LIN {X 0,Y 248.183,Z 542.153,A -85,B 0,C 180,E1 -18821.434,E2 -18821.434} C_VEL
LIN {X 0,Y 249.329,Z 538.255,A -85,B 0,C 180,E1 -18823.863,E2 -18823.863} C_VEL
LIN {X 0,Y 251.024,Z 533.251,A -85,B 0,C 180,E1 -18826.259,E2 -18826.259} C_VEL
LIN {X 0,Y 253.003,Z 526.994,A -85,B 0,C 180,E1 -18828.63,E2 -18828.63} C_VEL
LIN {X 0,Y 255.334,Z 519.2,A -85,B 0,C 180,E1 -18830.967,E2 -18830.967} C_VEL
LIN {X 0,Y 258.267,Z 509.494,A -85,B 0,C 180,E1 -18833.24,E2 -18833.24} C_VEL
LIN {X 0,Y 261.068,Z 499.47,A -85,B 0,C 180,E1 -18835.087,E2 -18835.087} C_VEL
LIN {X 0,Y 263.895,Z 488.136,A -85,B 0,C 180,E1 -18836.706,E2 -18836.706} C_VEL
LIN {X 0,Y 266.205,Z 477.049,A -85,B 0,C 180,E1 -18837.945,E2 -18837.945} C_VEL
LIN {X 0,Y 268.329,Z 464.711,A -85,B 0,C 180,E1 -18838.983,E2 -18838.983} C_VEL
LIN {X 0,Y 270.039,Z 451.206,A -85,B 0,C 180,E1 -18839.767,E2 -18839.767} C_VEL
LIN {X 0,Y 270.972,Z 437.637,A -85,B 0,C 180,E1 -18840.272,E2 -18840.272} C_VEL
LIN {X 0,Y 272.882,Z 389.185,A -85,B 0,C 180,E1 -18841.527,E2 -18841.527} C_VEL
LIN {X 0,Y 269.312,Z 367.58,A -85,B 0,C 180,E1 -18842.768,E2 -18842.768} C_VEL
LIN {X 0,Y 265.814,Z 359.147,A -85,B 0,C 180,E1 -18843.611,E2 -18843.611} C_VEL
LIN {X 0,Y 259.315,Z 346.028,A -85,B 0,C 180,E1 -18845.177,E2 -18845.177} C_VEL
LIN {X 0,Y 254.882,Z 337.632,A -85,B 0,C 180,E1 -18846.293,E2 -18846.293} C_VEL
LIN {X 0,Y 253.07,Z 333.942,A -85,B 0,C 180,E1 -18846.813,E2 -18846.813} C_VEL
LIN {X 0,Y 251.13,Z 326.758,A -85,B 0,C 180,E1 -18850.066,E2 -18850.066} C_VEL
LIN {X 0,Y 249.015,Z 319.468,A -85,B 0,C 180,E1 -18853.67,E2 -18853.67} C_VEL
LIN {X 0,Y 249.018,Z 319.462,A -85,B 0,C 180,E1 -18857.363,E2 -18857.363} C_VEL
LIN {X 0,Y 249.045,Z 319.458,A -85,B 0,C 180,E1 -18862.2,E2 -18862.2} C_VEL
LIN {X 0,Y 249.045,Z 319.455,A -85,B 0,C 180,E1 -18865.639,E2 -18865.639} C_VEL
LIN {X 0,Y 249.054,Z 319.453,A -85,B 0,C 180,E1 -18869.473,E2 -18869.473} C_VEL
LIN {X 0,Y 249.075,Z 319.451,A -85,B 0,C 180,E1 -18873.162,E2 -18873.162} C_VEL
LIN {X 0,Y 249.081,Z 319.451,A -85,B 0,C 180,E1 -18876.732,E2 -18876.732} C_VEL
LIN {X 0,Y 249.112,Z 319.451,A -85,B 0,C 180,E1 -18880.211,E2 -18880.211} C_VEL
LIN {X 0,Y 249.244,Z 319.437,A -85,B 0,C 180,E1 -18883.622,E2 -18883.622} C_VEL
LIN {X 0,Y 249.246,Z 319.432,A -85,B 0,C 180,E1 -18888.616,E2 -18888.616} C_VEL
LIN {X 0,Y 249.456,Z 319.407,A -85,B 0,C 180,E1 -18891.902,E2 -18891.902} C_VEL
LIN {X 0,Y 249.296,Z 319.417,A -85,B 0,C 180,E1 -18895.148,E2 -18895.148} C_VEL
LIN {X 0,Y 249.676,Z 319.367,A -85,B 0,C 180,E1 -18898.387,E2 -18898.387} C_VEL
LIN {X 0,Y 249.675,Z 319.379,A -85,B 0,C 180,E1 -18901.613,E2 -18901.613} C_VEL
LIN {X 0,Y 249.451,Z 319.402,A -85,B 0,C 180,E1 -18906.751,E2 -18906.751} C_VEL
LIN {X 0,Y 249.39,Z 319.416,A -85,B 0,C 180,E1 -18909.734,E2 -18909.734} C_VEL
LIN {X 0,Y 249.206,Z 319.442,A -85,B 0,C 180,E1 -18914.703,E2 -18914.703} C_VEL
LIN {X 0,Y 249.14,Z 319.449,A -85,B 0,C 180,E1 -18918.077,E2 -18918.077} C_VEL
LIN {X 0,Y 249.085,Z 319.452,A -85,B 0,C 180,E1 -18921.518,E2 -18921.518} C_VEL
LIN {X 0,Y 249.117,Z 319.447,A -85,B 0,C 180,E1 -18925.475,E2 -18925.475} C_VEL
LIN {X 0,Y 249.074,Z 319.45,A -85,B 0,C 180,E1 -18928.989,E2 -18928.989} C_VEL
LIN {X 0,Y 249.031,Z 319.457,A -85,B 0,C 180,E1 -18932.426,E2 -18932.426} C_VEL
LIN {X 0,Y 249.049,Z 319.461,A -85,B 0,C 180,E1 -18936.342,E2 -18936.342} C_VEL
LIN {X 0,Y 249.007,Z 319.463,A -85,B 0,C 180,E1 -18940.478,E2 -18940.478} C_VEL
LIN {X 0,Y 249.033,Z 319.491,A -85,B 0,C 180,E1 -18942.223,E2 -18942.223} C_VEL
LIN {X 0,Y 249.144,Z 320.169,A -85,B 0,C 180,E1 -18942.473,E2 -18942.473} C_VEL
LIN {X 0,Y 250.394,Z 322.834,A -85,B 0,C 180,E1 -18942.831,E2 -18942.831} C_VEL
LIN {X 0,Y 252.045,Z 324.832,A -85,B 0,C 180,E1 -18943.238,E2 -18943.238} C_VEL
LIN {X 0,Y 259.233,Z 336.696,A -85,B 0,C 180,E1 -18945.034,E2 -18945.034} C_VEL
LIN {X 0,Y 267.547,Z 352.366,A -85,B 0,C 180,E1 -18947.002,E2 -18947.002} C_VEL
LIN {X 0,Y 273.396,Z 365.109,A -85,B 0,C 180,E1 -18948.339,E2 -18948.339} C_VEL
LIN {X 0,Y 273.833,Z 366.225,A -85,B 0,C 180,E1 -18948.44,E2 -18948.44} C_VEL
LIN {X 0,Y 271.119,Z 427.277,A -85,B 0,C 180,E1 -18950.03,E2 -18950.03} C_VEL
LIN {X 0,Y 269.812,Z 441.335,A -85,B 0,C 180,E1 -18950.707,E2 -18950.707} C_VEL
LIN {X 0,Y 268.543,Z 451.318,A -85,B 0,C 180,E1 -18951.418,E2 -18951.418} C_VEL
LIN {X 0,Y 266.815,Z 462.787,A -85,B 0,C 180,E1 -18952.506,E2 -18952.506} C_VEL
LIN {X 0,Y 264.686,Z 473.393,A -85,B 0,C 180,E1 -18953.787,E2 -18953.787} C_VEL
LIN {X 0,Y 262.125,Z 484.416,A -85,B 0,C 180,E1 -18955.5,E2 -18955.5} C_VEL
LIN {X 0,Y 259.672,Z 493.358,A -85,B 0,C 180,E1 -18957.228,E2 -18957.228} C_VEL
LIN {X 0,Y 257.208,Z 501.535,A -85,B 0,C 180,E1 -18959.181,E2 -18959.181} C_VEL
LIN {X 0,Y 254.628,Z 509.489,A -85,B 0,C 180,E1 -18961.567,E2 -18961.567} C_VEL
LIN {X 0,Y 252.82,Z 514.863,A -85,B 0,C 180,E1 -18963.591,E2 -18963.591} C_VEL
LIN {X 0,Y 250.976,Z 520.041,A -85,B 0,C 180,E1 -18966.043,E2 -18966.043} C_VEL
LIN {X 0,Y 249.571,Z 524.019,A -85,B 0,C 180,E1 -18968.525,E2 -18968.525} C_VEL
LIN {X 0,Y 248.738,Z 526.048,A -85,B 0,C 180,E1 -18970.18,E2 -18970.18} C_VEL
LIN {X 0,Y 248.106,Z 527.649,A -85,B 0,C 180,E1 -18971.844,E2 -18971.844} C_VEL
LIN {X 0,Y 247.66,Z 528.827,A -85,B 0,C 180,E1 -18973.514,E2 -18973.514} C_VEL
LIN {X 0,Y 247.334,Z 529.546,A -85,B 0,C 180,E1 -18975.182,E2 -18975.182} C_VEL
LIN {X 0,Y 247.038,Z 529.872,A -85,B 0,C 180,E1 -18976.844,E2 -18976.844} C_VEL
LIN {X 0,Y 246.835,Z 529.809,A -85,B 0,C 180,E1 -18978.503,E2 -18978.503} C_VEL
LIN {X 0,Y 246.802,Z 529.34,A -85,B 0,C 180,E1 -18980.162,E2 -18980.162} C_VEL
LIN {X 0,Y 246.854,Z 528.434,A -85,B 0,C 180,E1 -18981.815,E2 -18981.815} C_VEL
LIN {X 0,Y 247.147,Z 526.179,A -85,B 0,C 180,E1 -18984.428,E2 -18984.428} C_VEL
LIN {X 0,Y 247.422,Z 523.28,A -85,B 0,C 180,E1 -18986.742,E2 -18986.742} C_VEL
LIN {X 0,Y 247.958,Z 519.177,A -85,B 0,C 180,E1 -18989.187,E2 -18989.187} C_VEL
LIN {X 0,Y 248.837,Z 512.912,A -85,B 0,C 180,E1 -18992.022,E2 -18992.022} C_VEL
LIN {X 0,Y 250.054,Z 506.085,A -85,B 0,C 180,E1 -18994.432,E2 -18994.432} C_VEL
LIN {X 0,Y 251.532,Z 497.568,A -85,B 0,C 180,E1 -18996.819,E2 -18996.819} C_VEL
LIN {X 0,Y 252.985,Z 488.83,A -85,B 0,C 180,E1 -18998.788,E2 -18998.788} C_VEL
LIN {X 0,Y 254.738,Z 478.068,A -85,B 0,C 180,E1 -19000.732,E2 -19000.732} C_VEL
LIN {X 0,Y 256.485,Z 467.223,A -85,B 0,C 180,E1 -19002.26,E2 -19002.26} C_VEL
LIN {X 0,Y 257.784,Z 457.077,A -85,B 0,C 180,E1 -19003.398,E2 -19003.398} C_VEL
LIN {X 0,Y 258.777,Z 445.087,A -85,B 0,C 180,E1 -19004.448,E2 -19004.448} C_VEL
LIN {X 0,Y 259.463,Z 433.861,A -85,B 0,C 180,E1 -19005.161,E2 -19005.161} C_VEL
LIN {X 0,Y 260.337,Z 420.826,A -85,B 0,C 180,E1 -19005.661,E2 -19005.661} C_VEL
LIN {X 0,Y 262.287,Z 353.407,A -85,B 0,C 180,E1 -19007.464,E2 -19007.464} C_VEL
LIN {X 0,Y 255.867,Z 335.25,A -85,B 0,C 180,E1 -19008.649,E2 -19008.649} C_VEL
LIN {X 0,Y 251.33,Z 324.687,A -85,B 0,C 180,E1 -19009.459,E2 -19009.459} C_VEL
LIN {X 0,Y 249.219,Z 320.139,A -85,B 0,C 180,E1 -19009.836,E2 -19009.836} C_VEL
LIN {X 0,Y 249.103,Z 319.457,A -85,B 0,C 180,E1 -19009.888,E2 -19009.888} C_VEL
LIN {X 0,Y 249.099,Z 319.453,A -85,B 0,C 180,E1 -19015.036,E2 -19015.036} C_VEL
LIN {X 0,Y 249.034,Z 319.462,A -85,B 0,C 180,E1 -19018.973,E2 -19018.973} C_VEL
LIN {X 0,Y 249.024,Z 319.465,A -85,B 0,C 180,E1 -19022.425,E2 -19022.425} C_VEL
LIN {X 0,Y 249.042,Z 319.463,A -85,B 0,C 180,E1 -19026.342,E2 -19026.342} C_VEL
LIN {X 0,Y 248.974,Z 319.47,A -85,B 0,C 180,E1 -19030.482,E2 -19030.482} C_VEL
LIN {X 0,Y 248.97,Z 319.463,A -85,B 0,C 180,E1 -19034.885,E2 -19034.885} C_VEL
LIN {X 0,Y 249.004,Z 319.468,A -85,B 0,C 180,E1 -19037.36,E2 -19037.36} C_VEL
LIN {X 0,Y 249.02,Z 319.455,A -85,B 0,C 180,E1 -19041.618,E2 -19041.618} C_VEL
LIN {X 0,Y 249.038,Z 319.463,A -85,B 0,C 180,E1 -19045.639,E2 -19045.639} C_VEL
LIN {X 0,Y 249.042,Z 319.45,A -85,B 0,C 180,E1 -19049.472,E2 -19049.472} C_VEL
LIN {X 0,Y 249.063,Z 319.457,A -85,B 0,C 180,E1 -19053.161,E2 -19053.161} C_VEL
LIN {X 0,Y 249.055,Z 319.457,A -85,B 0,C 180,E1 -19056.73,E2 -19056.73} C_VEL
LIN {X 0,Y 249.101,Z 319.443,A -85,B 0,C 180,E1 -19060.211,E2 -19060.211} C_VEL
LIN {X 0,Y 249.236,Z 319.437,A -85,B 0,C 180,E1 -19063.622,E2 -19063.622} C_VEL
LIN {X 0,Y 249.238,Z 319.427,A -85,B 0,C 180,E1 -19068.616,E2 -19068.616} C_VEL
LIN {X 0,Y 249.432,Z 319.405,A -85,B 0,C 180,E1 -19071.901,E2 -19071.901} C_VEL
LIN {X 0,Y 249.281,Z 319.431,A -85,B 0,C 180,E1 -19075.148,E2 -19075.148} C_VEL
LIN {X 0,Y 249.668,Z 319.378,A -85,B 0,C 180,E1 -19078.387,E2 -19078.387} C_VEL
LIN {X 0,Y 249.669,Z 319.371,A -85,B 0,C 180,E1 -19081.613,E2 -19081.613} C_VEL
LIN {X 0,Y 249.453,Z 319.413,A -85,B 0,C 180,E1 -19086.471,E2 -19086.471} C_VEL
LIN {X 0,Y 249.467,Z 319.408,A -85,B 0,C 180,E1 -19088.005,E2 -19088.005} C_VEL
LIN {X 0,Y 249.196,Z 319.446,A -85,B 0,C 180,E1 -19088.904,E2 -19088.904} C_VEL
LIN {X 0,Y 247.858,Z 319.618,A -85,B 0,C 180,E1 -19090.231,E2 -19090.231} C_VEL
LIN {X 0,Y 243.395,Z 320.175,A -85,B 0,C 180,E1 -19093.32,E2 -19093.32} C_VEL
LIN {X 0,Y 242.265,Z 320.31,A -85,B 0,C 180,E1 -19094.706,E2 -19094.706} C_VEL
LIN {X 0,Y 242.156,Z 320.32,A -85,B 0,C 180,E1 -19095.177,E2 -19095.177} C_VEL
LIN {X 0,Y 242.067,Z 320.33,A -85,B 0,C 180,E1 -19098.625,E2 -19098.625} C_VEL
LIN {X 0,Y 242.008,Z 320.336,A -85,B 0,C 180,E1 -19102.181,E2 -19102.181} C_VEL
LIN {X 0,Y 242.062,Z 320.329,A -85,B 0,C 180,E1 -19105.839,E2 -19105.839} C_VEL
LIN {X 0,Y 242.026,Z 320.336,A -85,B 0,C 180,E1 -19109.581,E2 -19109.581} C_VEL
LIN {X 0,Y 241.987,Z 320.343,A -85,B 0,C 180,E1 -19113.492,E2 -19113.492} C_VEL
LIN {X 0,Y 241.999,Z 320.344,A -85,B 0,C 180,E1 -19117.581,E2 -19117.581} C_VEL
LIN {X 0,Y 241.935,Z 320.351,A -85,B 0,C 180,E1 -19121.923,E2 -19121.923} C_VEL
LIN {X 0,Y 241.922,Z 320.35,A -85,B 0,C 180,E1 -19126.575,E2 -19126.575} C_VEL
LIN {X 0,Y 241.954,Z 320.347,A -85,B 0,C 180,E1 -19130.282,E2 -19130.282} C_VEL
LIN {X 0,Y 242.06,Z 320.442,A -85,B 0,C 180,E1 -19134.076,E2 -19134.076} C_VEL
LIN {X 0,Y 244.118,Z 330.064,A -85,B 0,C 180,E1 -19137.82,E2 -19137.82} C_VEL
LIN {X 0,Y 245.226,Z 335.144,A -85,B 0,C 180,E1 -19139.687,E2 -19139.687} C_VEL
LIN {X 0,Y 250.334,Z 348.902,A -85,B 0,C 180,E1 -19140.687,E2 -19140.687} C_VEL
LIN {X 0,Y 254.733,Z 384.139,A -85,B 0,C 180,E1 -19142.22,E2 -19142.22} C_VEL
LIN {X 0,Y 254.839,Z 390.528,A -85,B 0,C 180,E1 -19142.424,E2 -19142.424} C_VEL
LIN {X 0,Y 253.185,Z 443.682,A -85,B 0,C 180,E1 -19143.91,E2 -19143.91} C_VEL
LIN {X 0,Y 252.179,Z 457.01,A -85,B 0,C 180,E1 -19144.574,E2 -19144.574} C_VEL
LIN {X 0,Y 250.978,Z 469.25,A -85,B 0,C 180,E1 -19145.495,E2 -19145.495} C_VEL
LIN {X 0,Y 249.326,Z 481.555,A -85,B 0,C 180,E1 -19146.758,E2 -19146.758} C_VEL
LIN {X 0,Y 247.437,Z 493.191,A -85,B 0,C 180,E1 -19148.332,E2 -19148.332} C_VEL
LIN {X 0,Y 245.743,Z 503.799,A -85,B 0,C 180,E1 -19150.17,E2 -19150.17} C_VEL
LIN {X 0,Y 244.221,Z 512.882,A -85,B 0,C 180,E1 -19152.138,E2 -19152.138} C_VEL
LIN {X 0,Y 242.738,Z 521.525,A -85,B 0,C 180,E1 -19154.467,E2 -19154.467} C_VEL
LIN {X 0,Y 241.404,Z 528.956,A -85,B 0,C 180,E1 -19156.961,E2 -19156.961} C_VEL
LIN {X 0,Y 240.489,Z 535.778,A -85,B 0,C 180,E1 -19159.902,E2 -19159.902} C_VEL
LIN {X 0,Y 240.038,Z 540.265,A -85,B 0,C 180,E1 -19162.43,E2 -19162.43} C_VEL
LIN {X 0,Y 239.901,Z 543.655,A -85,B 0,C 180,E1 -19164.959,E2 -19164.959} C_VEL
LIN {X 0,Y 239.857,Z 545.33,A -85,B 0,C 180,E1 -19166.641,E2 -19166.641} C_VEL
LIN {X 0,Y 239.925,Z 546.599,A -85,B 0,C 180,E1 -19168.322,E2 -19168.322} C_VEL
LIN {X 0,Y 239.957,Z 547.461,A -85,B 0,C 180,E1 -19170.001,E2 -19170.001} C_VEL
LIN {X 0,Y 239.903,Z 547.878,A -85,B 0,C 180,E1 -19171.68,E2 -19171.68} C_VEL
LIN {X 0,Y 239.842,Z 547.532,A -85,B 0,C 180,E1 -19175.044,E2 -19175.044} C_VEL
LIN {X 0,Y 239.952,Z 546.786,A -85,B 0,C 180,E1 -19176.729,E2 -19176.729} C_VEL
LIN {X 0,Y 240.209,Z 545.617,A -85,B 0,C 180,E1 -19178.413,E2 -19178.413} C_VEL
LIN {X 0,Y 241.208,Z 542.034,A -85,B 0,C 180,E1 -19181.769,E2 -19181.769} C_VEL
LIN {X 0,Y 242.407,Z 538.187,A -85,B 0,C 180,E1 -19184.267,E2 -19184.267} C_VEL
LIN {X 0,Y 244.198,Z 533.239,A -85,B 0,C 180,E1 -19186.727,E2 -19186.727} C_VEL
LIN {X 0,Y 246.278,Z 527.041,A -85,B 0,C 180,E1 -19189.159,E2 -19189.159} C_VEL
LIN {X 0,Y 248.702,Z 519.35,A -85,B 0,C 180,E1 -19191.554,E2 -19191.554} C_VEL
LIN {X 0,Y 251.778,Z 509.726,A -85,B 0,C 180,E1 -19193.876,E2 -19193.876} C_VEL
LIN {X 0,Y 254.672,Z 499.819,A -85,B 0,C 180,E1 -19195.763,E2 -19195.763} C_VEL
LIN {X 0,Y 257.587,Z 488.668,A -85,B 0,C 180,E1 -19197.415,E2 -19197.415} C_VEL
LIN {X 0,Y 259.995,Z 477.769,A -85,B 0,C 180,E1 -19198.673,E2 -19198.673} C_VEL
LIN {X 0,Y 262.181,Z 465.736,A -85,B 0,C 180,E1 -19199.73,E2 -19199.73} C_VEL
LIN {X 0,Y 263.972,Z 452.813,A -85,B 0,C 180,E1 -19200.533,E2 -19200.533} C_VEL
LIN {X 0,Y 265.031,Z 439.193,A -85,B 0,C 180,E1 -19201.081,E2 -19201.081} C_VEL
LIN {X 0,Y 267.081,Z 390.218,A -85,B 0,C 180,E1 -19202.377,E2 -19202.377} C_VEL
LIN {X 0,Y 263.694,Z 369.628,A -85,B 0,C 180,E1 -19203.609,E2 -19203.609} C_VEL
LIN {X 0,Y 258.646,Z 358.428,A -85,B 0,C 180,E1 -19204.862,E2 -19204.862} C_VEL
LIN {X 0,Y 250.756,Z 342.788,A -85,B 0,C 180,E1 -19206.903,E2 -19206.903} C_VEL
LIN {X 0,Y 245.737,Z 333.591,A -85,B 0,C 180,E1 -19208.308,E2 -19208.308} C_VEL
LIN {X 0,Y 243.276,Z 324.826,A -85,B 0,C 180,E1 -19212.571,E2 -19212.571} C_VEL
LIN {X 0,Y 241.967,Z 320.342,A -85,B 0,C 180,E1 -19215,E2 -19215} C_VEL
LIN {X 0,Y 241.935,Z 320.345,A -85,B 0,C 180,E1 -19219.05,E2 -19219.05} C_VEL
LIN {X 0,Y 241.99,Z 320.335,A -85,B 0,C 180,E1 -19222.418,E2 -19222.418} C_VEL
LIN {X 0,Y 241.982,Z 320.334,A -85,B 0,C 180,E1 -19226.507,E2 -19226.507} C_VEL
LIN {X 0,Y 242.039,Z 320.331,A -85,B 0,C 180,E1 -19230.587,E2 -19230.587} C_VEL
LIN {X 0,Y 242.07,Z 320.327,A -85,B 0,C 180,E1 -19234.183,E2 -19234.183} C_VEL
LIN {X 0,Y 242.055,Z 320.33,A -85,B 0,C 180,E1 -19238.297,E2 -19238.297} C_VEL
LIN {X 0,Y 242.165,Z 320.318,A -85,B 0,C 180,E1 -19243.278,E2 -19243.278} C_VEL
LIN {X 0,Y 242.182,Z 320.312,A -85,B 0,C 180,E1 -19248.279,E2 -19248.279} C_VEL
LIN {X 0,Y 242.401,Z 320.283,A -85,B 0,C 180,E1 -19251.664,E2 -19251.664} C_VEL
LIN {X 0,Y 242.257,Z 320.293,A -85,B 0,C 180,E1 -19255.007,E2 -19255.007} C_VEL
LIN {X 0,Y 242.636,Z 320.244,A -85,B 0,C 180,E1 -19258.34,E2 -19258.34} C_VEL
LIN {X 0,Y 242.636,Z 320.256,A -85,B 0,C 180,E1 -19261.66,E2 -19261.66} C_VEL
LIN {X 0,Y 242.429,Z 320.277,A -85,B 0,C 180,E1 -19266.728,E2 -19266.728} C_VEL
LIN {X 0,Y 242.315,Z 320.298,A -85,B 0,C 180,E1 -19270.022,E2 -19270.022} C_VEL
LIN {X 0,Y 242.168,Z 320.317,A -85,B 0,C 180,E1 -19275.141,E2 -19275.141} C_VEL
LIN {X 0,Y 242.073,Z 320.333,A -85,B 0,C 180,E1 -19278.624,E2 -19278.624} C_VEL
LIN {X 0,Y 242.007,Z 320.337,A -85,B 0,C 180,E1 -19282.18,E2 -19282.18} C_VEL
LIN {X 0,Y 242.068,Z 320.328,A -85,B 0,C 180,E1 -19285.838,E2 -19285.838} C_VEL
LIN {X 0,Y 242.008,Z 320.336,A -85,B 0,C 180,E1 -19289.583,E2 -19289.583} C_VEL
LIN {X 0,Y 241.981,Z 320.34,A -85,B 0,C 180,E1 -19293.492,E2 -19293.492} C_VEL
LIN {X 0,Y 241.99,Z 320.335,A -85,B 0,C 180,E1 -19297.582,E2 -19297.582} C_VEL
LIN {X 0,Y 241.989,Z 320.45,A -85,B 0,C 180,E1 -19300.937,E2 -19300.937} C_VEL
LIN {X 0,Y 243.023,Z 323.277,A -85,B 0,C 180,E1 -19301.282,E2 -19301.282} C_VEL
LIN {X 0,Y 245.051,Z 325.678,A -85,B 0,C 180,E1 -19301.821,E2 -19301.821} C_VEL
LIN {X 0,Y 247.04,Z 328.858,A -85,B 0,C 180,E1 -19302.367,E2 -19302.367} C_VEL
LIN {X 0,Y 251.277,Z 335.458,A -85,B 0,C 180,E1 -19303.482,E2 -19303.482} C_VEL
LIN {X 0,Y 258.725,Z 348.635,A -85,B 0,C 180,E1 -19305.362,E2 -19305.362} C_VEL
LIN {X 0,Y 265.924,Z 363.342,A -85,B 0,C 180,E1 -19307.102,E2 -19307.102} C_VEL
LIN {X 0,Y 267.98,Z 368.129,A -85,B 0,C 180,E1 -19307.594,E2 -19307.594} C_VEL
LIN {X 0,Y 265.307,Z 427.111,A -85,B 0,C 180,E1 -19309.158,E2 -19309.158} C_VEL
LIN {X 0,Y 264.062,Z 440.542,A -85,B 0,C 180,E1 -19309.803,E2 -19309.803} C_VEL
LIN {X 0,Y 262.829,Z 450.168,A -85,B 0,C 180,E1 -19310.474,E2 -19310.474} C_VEL
LIN {X 0,Y 261.038,Z 461.61,A -85,B 0,C 180,E1 -19311.539,E2 -19311.539} C_VEL
LIN {X 0,Y 258.832,Z 472.452,A -85,B 0,C 180,E1 -19312.832,E2 -19312.832} C_VEL
LIN {X 0,Y 256.46,Z 482.659,A -85,B 0,C 180,E1 -19314.385,E2 -19314.385} C_VEL
LIN {X 0,Y 253.546,Z 492.855,A -85,B 0,C 180,E1 -19316.332,E2 -19316.332} C_VEL
LIN {X 0,Y 250.949,Z 501.161,A -85,B 0,C 180,E1 -19318.324,E2 -19318.324} C_VEL
LIN {X 0,Y 248.222,Z 509.261,A -85,B 0,C 180,E1 -19320.764,E2 -19320.764} C_VEL
LIN {X 0,Y 246.291,Z 514.701,A -85,B 0,C 180,E1 -19322.834,E2 -19322.834} C_VEL
LIN {X 0,Y 244.313,Z 519.986,A -85,B 0,C 180,E1 -19325.347,E2 -19325.347} C_VEL
LIN {X 0,Y 242.783,Z 524.049,A -85,B 0,C 180,E1 -19327.894,E2 -19327.894} C_VEL
LIN {X 0,Y 241.908,Z 526.125,A -85,B 0,C 180,E1 -19329.596,E2 -19329.596} C_VEL
LIN {X 0,Y 241.182,Z 527.762,A -85,B 0,C 180,E1 -19331.304,E2 -19331.304} C_VEL
LIN {X 0,Y 240.674,Z 528.983,A -85,B 0,C 180,E1 -19333.021,E2 -19333.021} C_VEL
LIN {X 0,Y 240.289,Z 529.791,A -85,B 0,C 180,E1 -19334.837,E2 -19334.837} C_VEL
LIN {X 0,Y 239.782,Z 530.094,A -85,B 0,C 180,E1 -19338.16,E2 -19338.16} C_VEL
LIN {X 0,Y 239.725,Z 529.675,A -85,B 0,C 180,E1 -19339.868,E2 -19339.868} C_VEL
LIN {X 0,Y 239.757,Z 528.821,A -85,B 0,C 180,E1 -19341.571,E2 -19341.571} C_VEL
LIN {X 0,Y 240.057,Z 526.383,A -85,B 0,C 180,E1 -19344.5,E2 -19344.5} C_VEL
LIN {X 0,Y 240.413,Z 522.57,A -85,B 0,C 180,E1 -19347.486,E2 -19347.486} C_VEL
LIN {X 0,Y 241.096,Z 518.172,A -85,B 0,C 180,E1 -19349.999,E2 -19349.999} C_VEL
LIN {X 0,Y 241.915,Z 512.599,A -85,B 0,C 180,E1 -19352.497,E2 -19352.497} C_VEL
LIN {X 0,Y 243.212,Z 505.624,A -85,B 0,C 180,E1 -19354.972,E2 -19354.972} C_VEL
LIN {X 0,Y 244.787,Z 496.898,A -85,B 0,C 180,E1 -19357.422,E2 -19357.422} C_VEL
LIN {X 0,Y 246.555,Z 486.993,A -85,B 0,C 180,E1 -19359.639,E2 -19359.639} C_VEL
LIN {X 0,Y 248.183,Z 476.907,A -85,B 0,C 180,E1 -19361.432,E2 -19361.432} C_VEL
LIN {X 0,Y 249.808,Z 467.238,A -85,B 0,C 180,E1 -19362.799,E2 -19362.799} C_VEL
LIN {X 0,Y 251.153,Z 457.027,A -85,B 0,C 180,E1 -19363.965,E2 -19363.965} C_VEL
LIN {X 0,Y 252.181,Z 444.941,A -85,B 0,C 180,E1 -19365.041,E2 -19365.041} C_VEL
LIN {X 0,Y 252.921,Z 433.539,A -85,B 0,C 180,E1 -19365.77,E2 -19365.77} C_VEL
LIN {X 0,Y 253.804,Z 420.407,A -85,B 0,C 180,E1 -19366.271,E2 -19366.271} C_VEL
LIN {X 0,Y 255.766,Z 354.635,A -85,B 0,C 180,E1 -19368.069,E2 -19368.069} C_VEL
LIN {X 0,Y 248.988,Z 335.878,A -85,B 0,C 180,E1 -19369.366,E2 -19369.366} C_VEL
LIN {X 0,Y 244.65,Z 326.267,A -85,B 0,C 180,E1 -19370.163,E2 -19370.163} C_VEL
LIN {X 0,Y 242.224,Z 321.153,A -85,B 0,C 180,E1 -19370.616,E2 -19370.616} C_VEL
LIN {X 0,Y 242.075,Z 320.333,A -85,B 0,C 180,E1 -19370.751,E2 -19370.751} C_VEL
LIN {X 0,Y 242.03,Z 320.333,A -85,B 0,C 180,E1 -19375.82,E2 -19375.82} C_VEL
LIN {X 0,Y 241.966,Z 320.341,A -85,B 0,C 180,E1 -19379.587,E2 -19379.587} C_VEL
LIN {X 0,Y 241.976,Z 320.342,A -85,B 0,C 180,E1 -19383.492,E2 -19383.492} C_VEL
LIN {X 0,Y 241.983,Z 320.337,A -85,B 0,C 180,E1 -19387.581,E2 -19387.581} C_VEL
LIN {X 0,Y 241.904,Z 320.35,A -85,B 0,C 180,E1 -19391.928,E2 -19391.928} C_VEL
LIN {X 0,Y 241.918,Z 320.346,A -85,B 0,C 180,E1 -19396.573,E2 -19396.573} C_VEL
LIN {X 0,Y 241.951,Z 320.337,A -85,B 0,C 180,E1 -19400.28,E2 -19400.28} C_VEL
LIN {X 0,Y 241.981,Z 320.339,A -85,B 0,C 180,E1 -19404.488,E2 -19404.488} C_VEL
LIN {X 0,Y 241.967,Z 320.335,A -85,B 0,C 180,E1 -19408.479,E2 -19408.479} C_VEL
LIN {X 0,Y 241.996,Z 320.336,A -85,B 0,C 180,E1 -19412.311,E2 -19412.311} C_VEL
LIN {X 0,Y 242.035,Z 320.334,A -85,B 0,C 180,E1 -19416.014,E2 -19416.014} C_VEL
LIN {X 0,Y 242.029,Z 320.322,A -85,B 0,C 180,E1 -19419.607,E2 -19419.607} C_VEL
LIN {X 0,Y 242.157,Z 320.317,A -85,B 0,C 180,E1 -19423.278,E2 -19423.278} C_VEL
LIN {X 0,Y 242.174,Z 320.308,A -85,B 0,C 180,E1 -19428.279,E2 -19428.279} C_VEL
LIN {X 0,Y 242.381,Z 320.281,A -85,B 0,C 180,E1 -19431.664,E2 -19431.664} C_VEL
LIN {X 0,Y 242.241,Z 320.308,A -85,B 0,C 180,E1 -19435.007,E2 -19435.007} C_VEL
LIN {X 0,Y 242.628,Z 320.254,A -85,B 0,C 180,E1 -19438.34,E2 -19438.34} C_VEL
LIN {X 0,Y 242.629,Z 320.247,A -85,B 0,C 180,E1 -19441.66,E2 -19441.66} C_VEL
LIN {X 0,Y 242.425,Z 320.287,A -85,B 0,C 180,E1 -19446.659,E2 -19446.659} C_VEL
LIN {X 0,Y 242.308,Z 320.29,A -85,B 0,C 180,E1 -19450.022,E2 -19450.022} C_VEL
LIN {X 0,Y 242.156,Z 320.32,A -85,B 0,C 180,E1 -19455.177,E2 -19455.177} C_VEL
LIN {X 0,Y 241.436,Z 320.412,A -85,B 0,C 180,E1 -19456.563,E2 -19456.563} C_VEL
LIN {X 0,Y 238.546,Z 320.77,A -85,B 0,C 180,E1 -19458.824,E2 -19458.824} C_VEL
LIN {X 0,Y 236.11,Z 321.075,A -85,B 0,C 180,E1 -19460.665,E2 -19460.665} C_VEL
LIN {X 0,Y 235.054,Z 321.202,A -85,B 0,C 180,E1 -19462.095,E2 -19462.095} C_VEL
LIN {X 0,Y 234.961,Z 321.214,A -85,B 0,C 180,E1 -19462.58,E2 -19462.58} C_VEL
LIN {X 0,Y 234.965,Z 321.215,A -85,B 0,C 180,E1 -19466.658,E2 -19466.658} C_VEL
LIN {X 0,Y 234.928,Z 321.22,A -85,B 0,C 180,E1 -19470.569,E2 -19470.569} C_VEL
LIN {X 0,Y 234.957,Z 321.218,A -85,B 0,C 180,E1 -19474.634,E2 -19474.634} C_VEL
LIN {X 0,Y 234.938,Z 321.223,A -85,B 0,C 180,E1 -19478.946,E2 -19478.946} C_VEL
LIN {X 0,Y 234.875,Z 321.232,A -85,B 0,C 180,E1 -19483.489,E2 -19483.489} C_VEL
LIN {X 0,Y 234.875,Z 321.228,A -85,B 0,C 180,E1 -19486.513,E2 -19486.513} C_VEL
LIN {X 0,Y 234.916,Z 321.223,A -85,B 0,C 180,E1 -19491.08,E2 -19491.08} C_VEL
LIN {X 0,Y 234.993,Z 321.308,A -85,B 0,C 180,E1 -19493.449,E2 -19493.449} C_VEL
LIN {X 0,Y 237.084,Z 330.909,A -85,B 0,C 180,E1 -19497.329,E2 -19497.329} C_VEL
LIN {X 0,Y 237.916,Z 334.744,A -85,B 0,C 180,E1 -19498.813,E2 -19498.813} C_VEL
LIN {X 0,Y 244.064,Z 350.961,A -85,B 0,C 180,E1 -19500.063,E2 -19500.063} C_VEL
LIN {X 0,Y 248.234,Z 384.797,A -85,B 0,C 180,E1 -19501.586,E2 -19501.586} C_VEL
LIN {X 0,Y 248.344,Z 390.664,A -85,B 0,C 180,E1 -19501.781,E2 -19501.781} C_VEL
LIN {X 0,Y 246.572,Z 444.278,A -85,B 0,C 180,E1 -19503.327,E2 -19503.327} C_VEL
LIN {X 0,Y 245.453,Z 458.087,A -85,B 0,C 180,E1 -19504.054,E2 -19504.054} C_VEL
LIN {X 0,Y 244.062,Z 470.999,A -85,B 0,C 180,E1 -19505.095,E2 -19505.095} C_VEL
LIN {X 0,Y 242.292,Z 483.589,A -85,B 0,C 180,E1 -19506.496,E2 -19506.496} C_VEL
LIN {X 0,Y 240.409,Z 494.805,A -85,B 0,C 180,E1 -19508.117,E2 -19508.117} C_VEL
LIN {X 0,Y 238.86,Z 503.892,A -85,B 0,C 180,E1 -19509.775,E2 -19509.775} C_VEL
LIN {X 0,Y 237.166,Z 513.76,A -85,B 0,C 180,E1 -19512.022,E2 -19512.022} C_VEL
LIN {X 0,Y 235.612,Z 522.247,A -85,B 0,C 180,E1 -19514.429,E2 -19514.429} C_VEL
LIN {X 0,Y 234.26,Z 529.502,A -85,B 0,C 180,E1 -19516.998,E2 -19516.998} C_VEL
LIN {X 0,Y 233.467,Z 535.286,A -85,B 0,C 180,E1 -19519.595,E2 -19519.595} C_VEL
LIN {X 0,Y 232.99,Z 539.827,A -85,B 0,C 180,E1 -19522.2,E2 -19522.2} C_VEL
LIN {X 0,Y 232.814,Z 543.461,A -85,B 0,C 180,E1 -19524.993,E2 -19524.993} C_VEL
LIN {X 0,Y 232.833,Z 546.256,A -85,B 0,C 180,E1 -19528.271,E2 -19528.271} C_VEL
LIN {X 0,Y 232.887,Z 547.145,A -85,B 0,C 180,E1 -19530.001,E2 -19530.001} C_VEL
LIN {X 0,Y 232.811,Z 547.602,A -85,B 0,C 180,E1 -19531.731,E2 -19531.731} C_VEL
LIN {X 0,Y 232.746,Z 547.299,A -85,B 0,C 180,E1 -19535.198,E2 -19535.198} C_VEL
LIN {X 0,Y 232.889,Z 546.576,A -85,B 0,C 180,E1 -19536.934,E2 -19536.934} C_VEL
LIN {X 0,Y 233.179,Z 545.452,A -85,B 0,C 180,E1 -19538.668,E2 -19538.668} C_VEL
LIN {X 0,Y 234.244,Z 541.917,A -85,B 0,C 180,E1 -19542.124,E2 -19542.124} C_VEL
LIN {X 0,Y 235.51,Z 538.121,A -85,B 0,C 180,E1 -19544.695,E2 -19544.695} C_VEL
LIN {X 0,Y 237.377,Z 533.227,A -85,B 0,C 180,E1 -19547.222,E2 -19547.222} C_VEL
LIN {X 0,Y 239.579,Z 527.088,A -85,B 0,C 180,E1 -19549.716,E2 -19549.716} C_VEL
LIN {X 0,Y 242.107,Z 519.486,A -85,B 0,C 180,E1 -19552.172,E2 -19552.172} C_VEL
LIN {X 0,Y 245.322,Z 509.959,A -85,B 0,C 180,E1 -19554.545,E2 -19554.545} C_VEL
LIN {X 0,Y 248.299,Z 500.152,A -85,B 0,C 180,E1 -19556.475,E2 -19556.475} C_VEL
LIN {X 0,Y 251.324,Z 489.2,A -85,B 0,C 180,E1 -19558.158,E2 -19558.158} C_VEL
LIN {X 0,Y 254.18,Z 476.739,A -85,B 0,C 180,E1 -19559.62,E2 -19559.62} C_VEL
LIN {X 0,Y 256.48,Z 464.484,A -85,B 0,C 180,E1 -19560.688,E2 -19560.688} C_VEL
LIN {X 0,Y 258.288,Z 451.307,A -85,B 0,C 180,E1 -19561.487,E2 -19561.487} C_VEL
LIN {X 0,Y 259.31,Z 437.77,A -85,B 0,C 180,E1 -19562.021,E2 -19562.021} C_VEL
LIN {X 0,Y 261.352,Z 391.36,A -85,B 0,C 180,E1 -19563.263,E2 -19563.263} C_VEL
LIN {X 0,Y 258.362,Z 372.643,A -85,B 0,C 180,E1 -19564.416,E2 -19564.416} C_VEL
LIN {X 0,Y 252.414,Z 359.506,A -85,B 0,C 180,E1 -19565.966,E2 -19565.966} C_VEL
LIN {X 0,Y 245.886,Z 346.665,A -85,B 0,C 180,E1 -19567.741,E2 -19567.741} C_VEL
LIN {X 0,Y 240.813,Z 337.631,A -85,B 0,C 180,E1 -19569.188,E2 -19569.188} C_VEL
LIN {X 0,Y 238.396,Z 333.187,A -85,B 0,C 180,E1 -19569.96,E2 -19569.96} C_VEL
LIN {X 0,Y 236.36,Z 326.119,A -85,B 0,C 180,E1 -19573.602,E2 -19573.602} C_VEL
LIN {X 0,Y 234.901,Z 321.222,A -85,B 0,C 180,E1 -19576.398,E2 -19576.398} C_VEL
LIN {X 0,Y 234.92,Z 321.221,A -85,B 0,C 180,E1 -19581.079,E2 -19581.079} C_VEL
LIN {X 0,Y 234.932,Z 321.214,A -85,B 0,C 180,E1 -19585.362,E2 -19585.362} C_VEL
LIN {X 0,Y 234.934,Z 321.212,A -85,B 0,C 180,E1 -19589.432,E2 -19589.432} C_VEL
LIN {X 0,Y 234.996,Z 321.205,A -85,B 0,C 180,E1 -19593.794,E2 -19593.794} C_VEL
LIN {X 0,Y 235.013,Z 321.21,A -85,B 0,C 180,E1 -19598.97,E2 -19598.97} C_VEL
LIN {X 0,Y 235.098,Z 321.197,A -85,B 0,C 180,E1 -19603.059,E2 -19603.059} C_VEL
LIN {X 0,Y 235.116,Z 321.194,A -85,B 0,C 180,E1 -19607.922,E2 -19607.922} C_VEL
LIN {X 0,Y 235.332,Z 321.162,A -85,B 0,C 180,E1 -19611.412,E2 -19611.412} C_VEL
LIN {X 0,Y 235.394,Z 321.154,A -85,B 0,C 180,E1 -19613.141,E2 -19613.141} C_VEL
LIN {X 0,Y 235.596,Z 321.121,A -85,B 0,C 180,E1 -19618.29,E2 -19618.29} C_VEL
LIN {X 0,Y 235.596,Z 321.132,A -85,B 0,C 180,E1 -19621.709,E2 -19621.709} C_VEL
LIN {X 0,Y 235.405,Z 321.152,A -85,B 0,C 180,E1 -19626.858,E2 -19626.858} C_VEL
LIN {X 0,Y 235.239,Z 321.181,A -85,B 0,C 180,E1 -19630.326,E2 -19630.326} C_VEL
LIN {X 0,Y 235.115,Z 321.192,A -85,B 0,C 180,E1 -19635.606,E2 -19635.606} C_VEL
LIN {X 0,Y 235.009,Z 321.21,A -85,B 0,C 180,E1 -19639.205,E2 -19639.205} C_VEL
LIN {X 0,Y 234.953,Z 321.218,A -85,B 0,C 180,E1 -19642.883,E2 -19642.883} C_VEL
LIN {X 0,Y 234.968,Z 321.215,A -85,B 0,C 180,E1 -19646.657,E2 -19646.657} C_VEL
LIN {X 0,Y 234.923,Z 321.216,A -85,B 0,C 180,E1 -19650.569,E2 -19650.569} C_VEL
LIN {X 0,Y 234.931,Z 321.212,A -85,B 0,C 180,E1 -19654.638,E2 -19654.638} C_VEL
LIN {X 0,Y 234.945,Z 321.395,A -85,B 0,C 180,E1 -19659.315,E2 -19659.315} C_VEL
LIN {X 0,Y 235.96,Z 324.127,A -85,B 0,C 180,E1 -19659.68,E2 -19659.68} C_VEL
LIN {X 0,Y 238.083,Z 326.588,A -85,B 0,C 180,E1 -19660.289,E2 -19660.289} C_VEL
LIN {X 0,Y 240.201,Z 329.895,A -85,B 0,C 180,E1 -19660.915,E2 -19660.915} C_VEL
LIN {X 0,Y 241.677,Z 332.113,A -85,B 0,C 180,E1 -19661.337,E2 -19661.337} C_VEL
LIN {X 0,Y 246.279,Z 338.984,A -85,B 0,C 180,E1 -19662.598,E2 -19662.598} C_VEL
LIN {X 0,Y 254.183,Z 353.254,A -85,B 0,C 180,E1 -19664.695,E2 -19664.695} C_VEL
LIN {X 0,Y 261.074,Z 367.556,A -85,B 0,C 180,E1 -19666.432,E2 -19666.432} C_VEL
LIN {X 0,Y 262.218,Z 370.187,A -85,B 0,C 180,E1 -19666.717,E2 -19666.717} C_VEL
LIN {X 0,Y 259.481,Z 428.094,A -85,B 0,C 180,E1 -19668.292,E2 -19668.292} C_VEL
LIN {X 0,Y 258.135,Z 441.637,A -85,B 0,C 180,E1 -19668.966,E2 -19668.966} C_VEL
LIN {X 0,Y 256.684,Z 452.166,A -85,B 0,C 180,E1 -19669.74,E2 -19669.74} C_VEL
LIN {X 0,Y 254.759,Z 463.651,A -85,B 0,C 180,E1 -19670.872,E2 -19670.872} C_VEL
LIN {X 0,Y 252.409,Z 474.352,A -85,B 0,C 180,E1 -19672.225,E2 -19672.225} C_VEL
LIN {X 0,Y 249.63,Z 485.293,A -85,B 0,C 180,E1 -19674.005,E2 -19674.005} C_VEL
LIN {X 0,Y 246.698,Z 495.054,A -85,B 0,C 180,E1 -19675.999,E2 -19675.999} C_VEL
LIN {X 0,Y 243.757,Z 503.743,A -85,B 0,C 180,E1 -19678.252,E2 -19678.252} C_VEL
LIN {X 0,Y 240.791,Z 511.887,A -85,B 0,C 180,E1 -19680.966,E2 -19680.966} C_VEL
LIN {X 0,Y 238.335,Z 518.275,A -85,B 0,C 180,E1 -19683.747,E2 -19683.747} C_VEL
LIN {X 0,Y 236.519,Z 522.802,A -85,B 0,C 180,E1 -19686.35,E2 -19686.35} C_VEL
LIN {X 0,Y 235.086,Z 526.203,A -85,B 0,C 180,E1 -19688.976,E2 -19688.976} C_VEL
LIN {X 0,Y 234.286,Z 527.876,A -85,B 0,C 180,E1 -19690.732,E2 -19690.732} C_VEL
LIN {X 0,Y 233.705,Z 529.133,A -85,B 0,C 180,E1 -19692.498,E2 -19692.498} C_VEL
LIN {X 0,Y 233.233,Z 530.078,A -85,B 0,C 180,E1 -19694.634,E2 -19694.634} C_VEL
LIN {X 0,Y 232.742,Z 530.378,A -85,B 0,C 180,E1 -19697.796,E2 -19697.796} C_VEL
LIN {X 0,Y 232.644,Z 529.993,A -85,B 0,C 180,E1 -19699.556,E2 -19699.556} C_VEL
LIN {X 0,Y 232.648,Z 529.207,A -85,B 0,C 180,E1 -19701.312,E2 -19701.312} C_VEL
LIN {X 0,Y 232.976,Z 526.608,A -85,B 0,C 180,E1 -19704.553,E2 -19704.553} C_VEL
LIN {X 0,Y 233.323,Z 523.094,A -85,B 0,C 180,E1 -19707.409,E2 -19707.409} C_VEL
LIN {X 0,Y 234.009,Z 518.773,A -85,B 0,C 180,E1 -19709.999,E2 -19709.999} C_VEL
LIN {X 0,Y 234.84,Z 513.285,A -85,B 0,C 180,E1 -19712.572,E2 -19712.572} C_VEL
LIN {X 0,Y 236.149,Z 506.424,A -85,B 0,C 180,E1 -19715.121,E2 -19715.121} C_VEL
LIN {X 0,Y 237.791,Z 497.84,A -85,B 0,C 180,E1 -19717.642,E2 -19717.642} C_VEL
LIN {X 0,Y 239.368,Z 489.051,A -85,B 0,C 180,E1 -19719.718,E2 -19719.718} C_VEL
LIN {X 0,Y 241.274,Z 478.222,A -85,B 0,C 180,E1 -19721.764,E2 -19721.764} C_VEL
LIN {X 0,Y 243.17,Z 467.244,A -85,B 0,C 180,E1 -19723.367,E2 -19723.367} C_VEL
LIN {X 0,Y 244.543,Z 456.975,A -85,B 0,C 180,E1 -19724.563,E2 -19724.563} C_VEL
LIN {X 0,Y 245.599,Z 444.8,A -85,B 0,C 180,E1 -19725.667,E2 -19725.667} C_VEL
LIN {X 0,Y 246.41,Z 433.217,A -85,B 0,C 180,E1 -19726.411,E2 -19726.411} C_VEL
LIN {X 0,Y 247.256,Z 420.713,A -85,B 0,C 180,E1 -19726.892,E2 -19726.892} C_VEL
LIN {X 0,Y 249.207,Z 355.997,A -85,B 0,C 180,E1 -19728.71,E2 -19728.71} C_VEL
LIN {X 0,Y 243.057,Z 338.927,A -85,B 0,C 180,E1 -19729.939,E2 -19729.939} C_VEL
LIN {X 0,Y 238.909,Z 329.753,A -85,B 0,C 180,E1 -19730.732,E2 -19730.732} C_VEL
LIN {X 0,Y 235.121,Z 321.977,A -85,B 0,C 180,E1 -19731.463,E2 -19731.463} C_VEL
LIN {X 0,Y 235,Z 321.212,A -85,B 0,C 180,E1 -19731.548,E2 -19731.548} C_VEL
LIN {X 0,Y 234.966,Z 321.211,A -85,B 0,C 180,E1 -19736.192,E2 -19736.192} C_VEL
LIN {X 0,Y 234.896,Z 321.223,A -85,B 0,C 180,E1 -19740.571,E2 -19740.571} C_VEL
LIN {X 0,Y 234.926,Z 321.222,A -85,B 0,C 180,E1 -19744.637,E2 -19744.637} C_VEL
LIN {X 0,Y 234.908,Z 321.218,A -85,B 0,C 180,E1 -19748.934,E2 -19748.934} C_VEL
LIN {X 0,Y 234.853,Z 321.221,A -85,B 0,C 180,E1 -19753.492,E2 -19753.492} C_VEL
LIN {X 0,Y 234.871,Z 321.224,A -85,B 0,C 180,E1 -19756.51,E2 -19756.51} C_VEL
LIN {X 0,Y 234.912,Z 321.211,A -85,B 0,C 180,E1 -19761.078,E2 -19761.078} C_VEL
LIN {X 0,Y 234.924,Z 321.222,A -85,B 0,C 180,E1 -19765.361,E2 -19765.361} C_VEL
LIN {X 0,Y 234.917,Z 321.208,A -85,B 0,C 180,E1 -19769.43,E2 -19769.43} C_VEL
LIN {X 0,Y 234.988,Z 321.215,A -85,B 0,C 180,E1 -19773.794,E2 -19773.794} C_VEL
LIN {X 0,Y 234.991,Z 321.2,A -85,B 0,C 180,E1 -19778.968,E2 -19778.968} C_VEL
LIN {X 0,Y 235.09,Z 321.197,A -85,B 0,C 180,E1 -19783.059,E2 -19783.059} C_VEL
LIN {X 0,Y 235.108,Z 321.19,A -85,B 0,C 180,E1 -19787.922,E2 -19787.922} C_VEL
LIN {X 0,Y 235.315,Z 321.159,A -85,B 0,C 180,E1 -19791.412,E2 -19791.412} C_VEL
LIN {X 0,Y 235.353,Z 321.163,A -85,B 0,C 180,E1 -19793.14,E2 -19793.14} C_VEL
LIN {X 0,Y 235.588,Z 321.131,A -85,B 0,C 180,E1 -19798.291,E2 -19798.291} C_VEL
LIN {X 0,Y 235.589,Z 321.124,A -85,B 0,C 180,E1 -19801.71,E2 -19801.71} C_VEL
LIN {X 0,Y 235.396,Z 321.161,A -85,B 0,C 180,E1 -19806.859,E2 -19806.859} C_VEL
LIN {X 0,Y 235.232,Z 321.169,A -85,B 0,C 180,E1 -19810.327,E2 -19810.327} C_VEL
LIN {X 0,Y 235.106,Z 321.197,A -85,B 0,C 180,E1 -19815.607,E2 -19815.607} C_VEL
LIN {X 0,Y 235.003,Z 321.212,A -85,B 0,C 180,E1 -19819.206,E2 -19819.206} C_VEL
LIN {X 0,Y 234.961,Z 321.214,A -85,B 0,C 180,E1 -19822.58,E2 -19822.58} C_VEL
LIN {X 0,Y 234.271,Z 321.305,A -85,B 0,C 180,E1 -19824.011,E2 -19824.011} C_VEL
LIN {X 0,Y 231.412,Z 321.661,A -85,B 0,C 180,E1 -19826.346,E2 -19826.346} C_VEL
LIN {X 0,Y 229.003,Z 321.959,A -85,B 0,C 180,E1 -19828.25,E2 -19828.25} C_VEL
LIN {X 0,Y 227.982,Z 322.085,A -85,B 0,C 180,E1 -19829.728,E2 -19829.728} C_VEL
LIN {X 0,Y 227.904,Z 322.094,A -85,B 0,C 180,E1 -19830.228,E2 -19830.228} C_VEL
LIN {X 0,Y 227.886,Z 322.1,A -85,B 0,C 180,E1 -19833.719,E2 -19833.719} C_VEL
LIN {X 0,Y 227.866,Z 322.103,A -85,B 0,C 180,E1 -19838.087,E2 -19838.087} C_VEL
LIN {X 0,Y 227.805,Z 322.111,A -85,B 0,C 180,E1 -19842.744,E2 -19842.744} C_VEL
LIN {X 0,Y 227.803,Z 322.111,A -85,B 0,C 180,E1 -19847.258,E2 -19847.258} C_VEL
LIN {X 0,Y 227.854,Z 322.104,A -85,B 0,C 180,E1 -19851.913,E2 -19851.913} C_VEL
LIN {X 0,Y 227.906,Z 322.245,A -85,B 0,C 180,E1 -19852.808,E2 -19852.808} C_VEL
LIN {X 0,Y 229.999,Z 331.326,A -85,B 0,C 180,E1 -19856.633,E2 -19856.633} C_VEL
LIN {X 0,Y 230.669,Z 334.691,A -85,B 0,C 180,E1 -19857.897,E2 -19857.897} C_VEL
LIN {X 0,Y 236.963,Z 350.703,A -85,B 0,C 180,E1 -19859.229,E2 -19859.229} C_VEL
LIN {X 0,Y 238.028,Z 354.445,A -85,B 0,C 180,E1 -19859.481,E2 -19859.481} C_VEL
LIN {X 0,Y 241.971,Z 388.075,A -85,B 0,C 180,E1 -19861.025,E2 -19861.025} C_VEL
LIN {X 0,Y 240.081,Z 443.738,A -85,B 0,C 180,E1 -19862.664,E2 -19862.664} C_VEL
LIN {X 0,Y 238.914,Z 457.634,A -85,B 0,C 180,E1 -19863.406,E2 -19863.406} C_VEL
LIN {X 0,Y 237.471,Z 470.612,A -85,B 0,C 180,E1 -19864.472,E2 -19864.472} C_VEL
LIN {X 0,Y 235.744,Z 482.425,A -85,B 0,C 180,E1 -19865.802,E2 -19865.802} C_VEL
LIN {X 0,Y 233.754,Z 493.807,A -85,B 0,C 180,E1 -19867.461,E2 -19867.461} C_VEL
LIN {X 0,Y 231.968,Z 504.072,A -85,B 0,C 180,E1 -19869.379,E2 -19869.379} C_VEL
LIN {X 0,Y 230.278,Z 513.392,A -85,B 0,C 180,E1 -19871.566,E2 -19871.566} C_VEL
LIN {X 0,Y 228.698,Z 521.594,A -85,B 0,C 180,E1 -19873.945,E2 -19873.945} C_VEL
LIN {X 0,Y 227.311,Z 528.924,A -85,B 0,C 180,E1 -19876.593,E2 -19876.593} C_VEL
LIN {X 0,Y 226.458,Z 534.787,A -85,B 0,C 180,E1 -19879.27,E2 -19879.27} C_VEL
LIN {X 0,Y 225.917,Z 539.384,A -85,B 0,C 180,E1 -19881.954,E2 -19881.954} C_VEL
LIN {X 0,Y 225.712,Z 543.367,A -85,B 0,C 180,E1 -19885.13,E2 -19885.13} C_VEL
LIN {X 0,Y 225.743,Z 545.913,A -85,B 0,C 180,E1 -19888.217,E2 -19888.217} C_VEL
LIN {X 0,Y 225.819,Z 546.825,A -85,B 0,C 180,E1 -19890.001,E2 -19890.001} C_VEL
LIN {X 0,Y 225.721,Z 547.323,A -85,B 0,C 180,E1 -19891.785,E2 -19891.785} C_VEL
LIN {X 0,Y 225.654,Z 547.067,A -85,B 0,C 180,E1 -19895.362,E2 -19895.362} C_VEL
LIN {X 0,Y 226.136,Z 545.279,A -85,B 0,C 180,E1 -19898.94,E2 -19898.94} C_VEL
LIN {X 0,Y 226.598,Z 543.748,A -85,B 0,C 180,E1 -19900.726,E2 -19900.726} C_VEL
LIN {X 0,Y 227.628,Z 540.684,A -85,B 0,C 180,E1 -19903.39,E2 -19903.39} C_VEL
LIN {X 0,Y 229.226,Z 536.589,A -85,B 0,C 180,E1 -19906.019,E2 -19906.019} C_VEL
LIN {X 0,Y 231.663,Z 530.341,A -85,B 0,C 180,E1 -19909.034,E2 -19909.034} C_VEL
LIN {X 0,Y 234.085,Z 523.695,A -85,B 0,C 180,E1 -19911.533,E2 -19911.533} C_VEL
LIN {X 0,Y 236.602,Z 516.69,A -85,B 0,C 180,E1 -19913.642,E2 -19913.642} C_VEL
LIN {X 0,Y 239.507,Z 508.424,A -85,B 0,C 180,E1 -19915.647,E2 -19915.647} C_VEL
LIN {X 0,Y 242.645,Z 498.328,A -85,B 0,C 180,E1 -19917.609,E2 -19917.609} C_VEL
LIN {X 0,Y 245.867,Z 486.915,A -85,B 0,C 180,E1 -19919.309,E2 -19919.309} C_VEL
LIN {X 0,Y 248.393,Z 475.739,A -85,B 0,C 180,E1 -19920.617,E2 -19920.617} C_VEL
LIN {X 0,Y 250.852,Z 463.159,A -85,B 0,C 180,E1 -19921.69,E2 -19921.69} C_VEL
LIN {X 0,Y 252.601,Z 450.107,A -85,B 0,C 180,E1 -19922.479,E2 -19922.479} C_VEL
LIN {X 0,Y 253.646,Z 437.005,A -85,B 0,C 180,E1 -19922.982,E2 -19922.982} C_VEL
LIN {X 0,Y 255.696,Z 392.406,A -85,B 0,C 180,E1 -19924.191,E2 -19924.191} C_VEL
LIN {X 0,Y 253.049,Z 375.57,A -85,B 0,C 180,E1 -19925.265,E2 -19925.265} C_VEL
LIN {X 0,Y 246.135,Z 360.339,A -85,B 0,C 180,E1 -19927.167,E2 -19927.167} C_VEL
LIN {X 0,Y 239.417,Z 347.26,A -85,B 0,C 180,E1 -19929.112,E2 -19929.112} C_VEL
LIN {X 0,Y 233.544,Z 337.319,A -85,B 0,C 180,E1 -19930.901,E2 -19930.901} C_VEL
LIN {X 0,Y 231.036,Z 332.863,A -85,B 0,C 180,E1 -19931.734,E2 -19931.734} C_VEL
LIN {X 0,Y 229.209,Z 326.652,A -85,B 0,C 180,E1 -19935.152,E2 -19935.152} C_VEL
LIN {X 0,Y 227.817,Z 322.104,A -85,B 0,C 180,E1 -19937.908,E2 -19937.908} C_VEL
LIN {X 0,Y 227.846,Z 322.1,A -85,B 0,C 180,E1 -19941.909,E2 -19941.909} C_VEL
LIN {X 0,Y 227.881,Z 322.09,A -85,B 0,C 180,E1 -19946.377,E2 -19946.377} C_VEL
LIN {X 0,Y 227.921,Z 322.088,A -85,B 0,C 180,E1 -19950.438,E2 -19950.438} C_VEL
LIN {X 0,Y 227.931,Z 322.09,A -85,B 0,C 180,E1 -19954.426,E2 -19954.426} C_VEL
LIN {X 0,Y 227.964,Z 322.084,A -85,B 0,C 180,E1 -19958.287,E2 -19958.287} C_VEL
LIN {X 0,Y 228.036,Z 322.076,A -85,B 0,C 180,E1 -19962.826,E2 -19962.826} C_VEL
LIN {X 0,Y 228.074,Z 322.071,A -85,B 0,C 180,E1 -19967.543,E2 -19967.543} C_VEL
LIN {X 0,Y 228.269,Z 322.04,A -85,B 0,C 180,E1 -19971.144,E2 -19971.144} C_VEL
LIN {X 0,Y 228.341,Z 322.035,A -85,B 0,C 180,E1 -19972.928,E2 -19972.928} C_VEL
LIN {X 0,Y 228.555,Z 321.998,A -85,B 0,C 180,E1 -19978.238,E2 -19978.238} C_VEL
LIN {X 0,Y 228.554,Z 322.008,A -85,B 0,C 180,E1 -19981.762,E2 -19981.762} C_VEL
LIN {X 0,Y 228.356,Z 322.028,A -85,B 0,C 180,E1 -19987.071,E2 -19987.071} C_VEL
LIN {X 0,Y 228.16,Z 322.06,A -85,B 0,C 180,E1 -19990.65,E2 -19990.65} C_VEL
LIN {X 0,Y 228.066,Z 322.075,A -85,B 0,C 180,E1 -19994.272,E2 -19994.272} C_VEL
LIN {X 0,Y 228.004,Z 322.081,A -85,B 0,C 180,E1 -19997.953,E2 -19997.953} C_VEL
LIN {X 0,Y 227.918,Z 322.093,A -85,B 0,C 180,E1 -20002.321,E2 -20002.321} C_VEL
LIN {X 0,Y 227.942,Z 322.09,A -85,B 0,C 180,E1 -20006.602,E2 -20006.602} C_VEL
LIN {X 0,Y 227.898,Z 322.094,A -85,B 0,C 180,E1 -20010.29,E2 -20010.29} C_VEL
LIN {X 0,Y 227.878,Z 322.095,A -85,B 0,C 180,E1 -20013.72,E2 -20013.72} C_VEL
LIN {X 0,Y 227.841,Z 322.097,A -85,B 0,C 180,E1 -20017.51,E2 -20017.51} C_VEL
LIN {X 0,Y 228.812,Z 324.903,A -85,B 0,C 180,E1 -20017.901,E2 -20017.901} C_VEL
LIN {X 0,Y 231.266,Z 327.736,A -85,B 0,C 180,E1 -20018.667,E2 -20018.667} C_VEL
LIN {X 0,Y 233.435,Z 330.987,A -85,B 0,C 180,E1 -20019.355,E2 -20019.355} C_VEL
LIN {X 0,Y 240.025,Z 340.618,A -85,B 0,C 180,E1 -20021.31,E2 -20021.31} C_VEL
LIN {X 0,Y 245.949,Z 350.77,A -85,B 0,C 180,E1 -20022.983,E2 -20022.983} C_VEL
LIN {X 0,Y 253.049,Z 364.688,A -85,B 0,C 180,E1 -20024.897,E2 -20024.897} C_VEL
LIN {X 0,Y 256.525,Z 372.346,A -85,B 0,C 180,E1 -20025.804,E2 -20025.804} C_VEL
LIN {X 0,Y 253.825,Z 427.703,A -85,B 0,C 180,E1 -20027.328,E2 -20027.328} C_VEL
LIN {X 0,Y 252.429,Z 441.554,A -85,B 0,C 180,E1 -20028.02,E2 -20028.02} C_VEL
LIN {X 0,Y 251.051,Z 451.284,A -85,B 0,C 180,E1 -20028.73,E2 -20028.73} C_VEL
LIN {X 0,Y 249.153,Z 462.425,A -85,B 0,C 180,E1 -20029.815,E2 -20029.815} C_VEL
LIN {X 0,Y 246.687,Z 473.475,A -85,B 0,C 180,E1 -20031.187,E2 -20031.187} C_VEL
LIN {X 0,Y 244.104,Z 483.566,A -85,B 0,C 180,E1 -20032.799,E2 -20032.799} C_VEL
LIN {X 0,Y 241.12,Z 493.135,A -85,B 0,C 180,E1 -20034.699,E2 -20034.699} C_VEL
LIN {X 0,Y 238.108,Z 501.94,A -85,B 0,C 180,E1 -20036.903,E2 -20036.903} C_VEL
LIN {X 0,Y 235.105,Z 509.986,A -85,B 0,C 180,E1 -20039.457,E2 -20039.457} C_VEL
LIN {X 0,Y 232.575,Z 516.35,A -85,B 0,C 180,E1 -20042.07,E2 -20042.07} C_VEL
LIN {X 0,Y 230.436,Z 521.37,A -85,B 0,C 180,E1 -20044.723,E2 -20044.723} C_VEL
LIN {X 0,Y 229.013,Z 524.738,A -85,B 0,C 180,E1 -20047.02,E2 -20047.02} C_VEL
LIN {X 0,Y 227.415,Z 527.99,A -85,B 0,C 180,E1 -20050.126,E2 -20050.126} C_VEL
LIN {X 0,Y 226.785,Z 529.281,A -85,B 0,C 180,E1 -20051.946,E2 -20051.946} C_VEL
LIN {X 0,Y 226.197,Z 530.36,A -85,B 0,C 180,E1 -20054.403,E2 -20054.403} C_VEL
LIN {X 0,Y 225.684,Z 530.664,A -85,B 0,C 180,E1 -20057.408,E2 -20057.408} C_VEL
LIN {X 0,Y 225.56,Z 529.573,A -85,B 0,C 180,E1 -20061.037,E2 -20061.037} C_VEL
LIN {X 0,Y 225.654,Z 528.397,A -85,B 0,C 180,E1 -20062.843,E2 -20062.843} C_VEL
LIN {X 0,Y 225.947,Z 526.32,A -85,B 0,C 180,E1 -20065.12,E2 -20065.12} C_VEL
LIN {X 0,Y 226.354,Z 522.355,A -85,B 0,C 180,E1 -20068.22,E2 -20068.22} C_VEL
LIN {X 0,Y 227.153,Z 517.732,A -85,B 0,C 180,E1 -20070.885,E2 -20070.885} C_VEL
LIN {X 0,Y 228.371,Z 510.771,A -85,B 0,C 180,E1 -20073.969,E2 -20073.969} C_VEL
LIN {X 0,Y 229.932,Z 503.231,A -85,B 0,C 180,E1 -20076.581,E2 -20076.581} C_VEL
LIN {X 0,Y 231.373,Z 495.544,A -85,B 0,C 180,E1 -20078.735,E2 -20078.735} C_VEL
LIN {X 0,Y 233.199,Z 486.148,A -85,B 0,C 180,E1 -20080.856,E2 -20080.856} C_VEL
LIN {X 0,Y 235.034,Z 475.727,A -85,B 0,C 180,E1 -20082.739,E2 -20082.739} C_VEL
LIN {X 0,Y 236.906,Z 465.649,A -85,B 0,C 180,E1 -20084.166,E2 -20084.166} C_VEL
LIN {X 0,Y 238.26,Z 453.978,A -85,B 0,C 180,E1 -20085.504,E2 -20085.504} C_VEL
LIN {X 0,Y 239.302,Z 441.21,A -85,B 0,C 180,E1 -20086.583,E2 -20086.583} C_VEL
LIN {X 0,Y 240.266,Z 427.978,A -85,B 0,C 180,E1 -20087.311,E2 -20087.311} C_VEL
LIN {X 0,Y 241.379,Z 403.187,A -85,B 0,C 180,E1 -20088.052,E2 -20088.052} C_VEL
LIN {X 0,Y 242.802,Z 357.676,A -85,B 0,C 180,E1 -20089.362,E2 -20089.362} C_VEL
LIN {X 0,Y 236.353,Z 339.98,A -85,B 0,C 180,E1 -20090.702,E2 -20090.702} C_VEL
LIN {X 0,Y 230.512,Z 327.92,A -85,B 0,C 180,E1 -20091.856,E2 -20091.856} C_VEL
LIN {X 0,Y 228.124,Z 323.051,A -85,B 0,C 180,E1 -20092.347,E2 -20092.347} C_VEL
LIN {X 0,Y 227.921,Z 322.094,A -85,B 0,C 180,E1 -20092.417,E2 -20092.417} C_VEL
LIN {X 0,Y 227.92,Z 322.088,A -85,B 0,C 180,E1 -20096.591,E2 -20096.591} C_VEL
LIN {X 0,Y 227.87,Z 322.098,A -85,B 0,C 180,E1 -20100.279,E2 -20100.279} C_VEL
LIN {X 0,Y 227.874,Z 322.098,A -85,B 0,C 180,E1 -20103.719,E2 -20103.719} C_VEL
LIN {X 0,Y 227.839,Z 322.098,A -85,B 0,C 180,E1 -20108.09,E2 -20108.09} C_VEL
LIN {X 0,Y 227.783,Z 322.107,A -85,B 0,C 180,E1 -20112.747,E2 -20112.747} C_VEL
LIN {X 0,Y 227.8,Z 322.11,A -85,B 0,C 180,E1 -20117.255,E2 -20117.255} C_VEL
LIN {X 0,Y 227.838,Z 322.091,A -85,B 0,C 180,E1 -20121.908,E2 -20121.908} C_VEL
LIN {X 0,Y 227.874,Z 322.096,A -85,B 0,C 180,E1 -20126.377,E2 -20126.377} C_VEL
LIN {X 0,Y 227.899,Z 322.081,A -85,B 0,C 180,E1 -20130.435,E2 -20130.435} C_VEL
LIN {X 0,Y 227.919,Z 322.093,A -85,B 0,C 180,E1 -20134.425,E2 -20134.425} C_VEL
LIN {X 0,Y 227.941,Z 322.078,A -85,B 0,C 180,E1 -20138.285,E2 -20138.285} C_VEL
LIN {X 0,Y 228.029,Z 322.076,A -85,B 0,C 180,E1 -20142.826,E2 -20142.826} C_VEL
LIN {X 0,Y 228.066,Z 322.071,A -85,B 0,C 180,E1 -20147.543,E2 -20147.543} C_VEL
LIN {X 0,Y 228.253,Z 322.038,A -85,B 0,C 180,E1 -20151.144,E2 -20151.144} C_VEL
LIN {X 0,Y 228.305,Z 322.041,A -85,B 0,C 180,E1 -20152.927,E2 -20152.927} C_VEL
LIN {X 0,Y 228.546,Z 322.008,A -85,B 0,C 180,E1 -20158.238,E2 -20158.238} C_VEL
LIN {X 0,Y 228.548,Z 322,A -85,B 0,C 180,E1 -20161.762,E2 -20161.762} C_VEL
LIN {X 0,Y 228.347,Z 322.038,A -85,B 0,C 180,E1 -20167.072,E2 -20167.072} C_VEL
LIN {X 0,Y 228.153,Z 322.048,A -85,B 0,C 180,E1 -20170.651,E2 -20170.651} C_VEL
LIN {X 0,Y 228.057,Z 322.073,A -85,B 0,C 180,E1 -20174.273,E2 -20174.273} C_VEL
LIN {X 0,Y 227.998,Z 322.08,A -85,B 0,C 180,E1 -20177.954,E2 -20177.954} C_VEL
LIN {X 0,Y 227.914,Z 322.091,A -85,B 0,C 180,E1 -20182.562,E2 -20182.562} C_VEL
LIN {X 0,Y 227.938,Z 322.09,A -85,B 0,C 180,E1 -20186.604,E2 -20186.604} C_VEL
LIN {X 0,Y 227.904,Z 322.094,A -85,B 0,C 180,E1 -20190.228,E2 -20190.228} C_VEL
LIN {X 0,Y 227.25,Z 322.179,A -85,B 0,C 180,E1 -20191.703,E2 -20191.703} C_VEL
LIN {X 0,Y 224.399,Z 322.536,A -85,B 0,C 180,E1 -20194.108,E2 -20194.108} C_VEL
LIN {X 0,Y 221.952,Z 322.839,A -85,B 0,C 180,E1 -20196.071,E2 -20196.071} C_VEL
LIN {X 0,Y 220.882,Z 322.975,A -85,B 0,C 180,E1 -20197.595,E2 -20197.595} C_VEL
LIN {X 0,Y 220.785,Z 322.98,A -85,B 0,C 180,E1 -20198.112,E2 -20198.112} C_VEL
LIN {X 0,Y 220.768,Z 322.988,A -85,B 0,C 180,E1 -20201.953,E2 -20201.953} C_VEL
LIN {X 0,Y 220.764,Z 322.988,A -85,B 0,C 180,E1 -20205.546,E2 -20205.546} C_VEL
LIN {X 0,Y 220.804,Z 322.981,A -85,B 0,C 180,E1 -20210.465,E2 -20210.465} C_VEL
LIN {X 0,Y 220.848,Z 323.072,A -85,B 0,C 180,E1 -20212.082,E2 -20212.082} C_VEL
LIN {X 0,Y 222.969,Z 332.317,A -85,B 0,C 180,E1 -20216.127,E2 -20216.127} C_VEL
LIN {X 0,Y 223.422,Z 334.391,A -85,B 0,C 180,E1 -20216.907,E2 -20216.907} C_VEL
LIN {X 0,Y 230.56,Z 352.303,A -85,B 0,C 180,E1 -20218.491,E2 -20218.491} C_VEL
LIN {X 0,Y 231.76,Z 356.205,A -85,B 0,C 180,E1 -20218.777,E2 -20218.777} C_VEL
LIN {X 0,Y 235.47,Z 387.911,A -85,B 0,C 180,E1 -20220.291,E2 -20220.291} C_VEL
LIN {X 0,Y 233.595,Z 443.151,A -85,B 0,C 180,E1 -20221.961,E2 -20221.961} C_VEL
LIN {X 0,Y 232.501,Z 456.4,A -85,B 0,C 180,E1 -20222.673,E2 -20222.673} C_VEL
LIN {X 0,Y 231.056,Z 469.156,A -85,B 0,C 180,E1 -20223.709,E2 -20223.709} C_VEL
LIN {X 0,Y 229.246,Z 481.258,A -85,B 0,C 180,E1 -20225.07,E2 -20225.07} C_VEL
LIN {X 0,Y 227.22,Z 492.814,A -85,B 0,C 180,E1 -20226.775,E2 -20226.775} C_VEL
LIN {X 0,Y 225.258,Z 503.23,A -85,B 0,C 180,E1 -20228.735,E2 -20228.735} C_VEL
LIN {X 0,Y 223.471,Z 512.101,A -85,B 0,C 180,E1 -20230.825,E2 -20230.825} C_VEL
LIN {X 0,Y 222.405,Z 518.101,A -85,B 0,C 180,E1 -20232.532,E2 -20232.532} C_VEL
LIN {X 0,Y 220.853,Z 526.083,A -85,B 0,C 180,E1 -20235.253,E2 -20235.253} C_VEL
LIN {X 0,Y 219.678,Z 532.437,A -85,B 0,C 180,E1 -20237.999,E2 -20237.999} C_VEL
LIN {X 0,Y 219.028,Z 537.49,A -85,B 0,C 180,E1 -20240.769,E2 -20240.769} C_VEL
LIN {X 0,Y 218.699,Z 541.386,A -85,B 0,C 180,E1 -20243.543,E2 -20243.543} C_VEL
LIN {X 0,Y 218.588,Z 544.231,A -85,B 0,C 180,E1 -20246.314,E2 -20246.314} C_VEL
LIN {X 0,Y 218.656,Z 545.57,A -85,B 0,C 180,E1 -20248.159,E2 -20248.159} C_VEL
LIN {X 0,Y 218.751,Z 546.505,A -85,B 0,C 180,E1 -20250.001,E2 -20250.001} C_VEL
LIN {X 0,Y 218.632,Z 547.035,A -85,B 0,C 180,E1 -20251.843,E2 -20251.843} C_VEL
LIN {X 0,Y 218.542,Z 547.049,A -85,B 0,C 180,E1 -20254.497,E2 -20254.497} C_VEL
LIN {X 0,Y 218.76,Z 546.156,A -85,B 0,C 180,E1 -20257.384,E2 -20257.384} C_VEL
LIN {X 0,Y 219.09,Z 545.094,A -85,B 0,C 180,E1 -20259.23,E2 -20259.23} C_VEL
LIN {X 0,Y 219.61,Z 543.608,A -85,B 0,C 180,E1 -20261.071,E2 -20261.071} C_VEL
LIN {X 0,Y 220.689,Z 540.593,A -85,B 0,C 180,E1 -20263.819,E2 -20263.819} C_VEL
LIN {X 0,Y 222.394,Z 536.55,A -85,B 0,C 180,E1 -20266.525,E2 -20266.525} C_VEL
LIN {X 0,Y 224.95,Z 530.366,A -85,B 0,C 180,E1 -20269.625,E2 -20269.625} C_VEL
LIN {X 0,Y 227.544,Z 523.66,A -85,B 0,C 180,E1 -20272.233,E2 -20272.233} C_VEL
LIN {X 0,Y 230.679,Z 515.369,A -85,B 0,C 180,E1 -20274.767,E2 -20274.767} C_VEL
LIN {X 0,Y 233.767,Z 506.867,A -85,B 0,C 180,E1 -20276.806,E2 -20276.806} C_VEL
LIN {X 0,Y 236.792,Z 497.567,A -85,B 0,C 180,E1 -20278.594,E2 -20278.594} C_VEL
LIN {X 0,Y 239.728,Z 487.47,A -85,B 0,C 180,E1 -20280.136,E2 -20280.136} C_VEL
LIN {X 0,Y 242.343,Z 476.49,A -85,B 0,C 180,E1 -20281.467,E2 -20281.467} C_VEL
LIN {X 0,Y 244.88,Z 464.311,A -85,B 0,C 180,E1 -20282.556,E2 -20282.556} C_VEL
LIN {X 0,Y 246.764,Z 451.401,A -85,B 0,C 180,E1 -20283.381,E2 -20283.381} C_VEL
LIN {X 0,Y 247.912,Z 438.295,A -85,B 0,C 180,E1 -20283.923,E2 -20283.923} C_VEL
LIN {X 0,Y 250.107,Z 393.985,A -85,B 0,C 180,E1 -20285.142,E2 -20285.142} C_VEL
LIN {X 0,Y 247.776,Z 378.431,A -85,B 0,C 180,E1 -20286.157,E2 -20286.157} C_VEL
LIN {X 0,Y 241.098,Z 363.664,A -85,B 0,C 180,E1 -20288.089,E2 -20288.089} C_VEL
LIN {X 0,Y 235.004,Z 351.727,A -85,B 0,C 180,E1 -20289.94,E2 -20289.94} C_VEL
LIN {X 0,Y 229.686,Z 342.474,A -85,B 0,C 180,E1 -20291.642,E2 -20291.642} C_VEL
LIN {X 0,Y 226.261,Z 336.916,A -85,B 0,C 180,E1 -20292.791,E2 -20292.791} C_VEL
LIN {X 0,Y 223.651,Z 332.443,A -85,B 0,C 180,E1 -20293.736,E2 -20293.736} C_VEL
LIN {X 0,Y 221.397,Z 325.065,A -85,B 0,C 180,E1 -20298.193,E2 -20298.193} C_VEL
LIN {X 0,Y 220.801,Z 322.974,A -85,B 0,C 180,E1 -20299.612,E2 -20299.612} C_VEL
LIN {X 0,Y 220.827,Z 322.97,A -85,B 0,C 180,E1 -20302.793,E2 -20302.793} C_VEL
LIN {X 0,Y 220.82,Z 322.974,A -85,B 0,C 180,E1 -20307.244,E2 -20307.244} C_VEL
LIN {X 0,Y 220.839,Z 322.977,A -85,B 0,C 180,E1 -20311.486,E2 -20311.486} C_VEL
LIN {X 0,Y 220.87,Z 322.972,A -85,B 0,C 180,E1 -20315.565,E2 -20315.565} C_VEL
LIN {X 0,Y 220.894,Z 322.969,A -85,B 0,C 180,E1 -20319.514,E2 -20319.514} C_VEL
LIN {X 0,Y 221.018,Z 322.953,A -85,B 0,C 180,E1 -20323.37,E2 -20323.37} C_VEL
LIN {X 0,Y 221.013,Z 322.948,A -85,B 0,C 180,E1 -20327.138,E2 -20327.138} C_VEL
LIN {X 0,Y 221.206,Z 322.917,A -85,B 0,C 180,E1 -20330.859,E2 -20330.859} C_VEL
LIN {X 0,Y 221.273,Z 322.916,A -85,B 0,C 180,E1 -20332.701,E2 -20332.701} C_VEL
LIN {X 0,Y 221.513,Z 322.876,A -85,B 0,C 180,E1 -20338.182,E2 -20338.182} C_VEL
LIN {X 0,Y 221.512,Z 322.884,A -85,B 0,C 180,E1 -20341.818,E2 -20341.818} C_VEL
LIN {X 0,Y 221.291,Z 322.906,A -85,B 0,C 180,E1 -20347.298,E2 -20347.298} C_VEL
LIN {X 0,Y 221.108,Z 322.937,A -85,B 0,C 180,E1 -20350.994,E2 -20350.994} C_VEL
LIN {X 0,Y 221.018,Z 322.944,A -85,B 0,C 180,E1 -20356.63,E2 -20356.63} C_VEL
LIN {X 0,Y 220.886,Z 322.961,A -85,B 0,C 180,E1 -20360.487,E2 -20360.487} C_VEL
LIN {X 0,Y 220.863,Z 322.963,A -85,B 0,C 180,E1 -20364.435,E2 -20364.435} C_VEL
LIN {X 0,Y 220.828,Z 322.966,A -85,B 0,C 180,E1 -20368.515,E2 -20368.515} C_VEL
LIN {X 0,Y 220.817,Z 322.973,A -85,B 0,C 180,E1 -20372.756,E2 -20372.756} C_VEL
LIN {X 0,Y 220.853,Z 323.099,A -85,B 0,C 180,E1 -20375.573,E2 -20375.573} C_VEL
LIN {X 0,Y 221.755,Z 325.664,A -85,B 0,C 180,E1 -20375.966,E2 -20375.966} C_VEL
LIN {X 0,Y 223.737,Z 327.852,A -85,B 0,C 180,E1 -20376.643,E2 -20376.643} C_VEL
LIN {X 0,Y 226.601,Z 332.06,A -85,B 0,C 180,E1 -20377.633,E2 -20377.633} C_VEL
LIN {X 0,Y 228.092,Z 334.118,A -85,B 0,C 180,E1 -20378.126,E2 -20378.126} C_VEL
LIN {X 0,Y 231.261,Z 338.687,A -85,B 0,C 180,E1 -20379.146,E2 -20379.146} C_VEL
LIN {X 0,Y 237.688,Z 348.337,A -85,B 0,C 180,E1 -20381.095,E2 -20381.095} C_VEL
LIN {X 0,Y 245.471,Z 362.922,A -85,B 0,C 180,E1 -20383.351,E2 -20383.351} C_VEL
LIN {X 0,Y 250.906,Z 374.529,A -85,B 0,C 180,E1 -20384.853,E2 -20384.853} C_VEL
LIN {X 0,Y 248.184,Z 428.06,A -85,B 0,C 180,E1 -20386.353,E2 -20386.353} C_VEL
LIN {X 0,Y 246.805,Z 441.41,A -85,B 0,C 180,E1 -20387.028,E2 -20387.028} C_VEL
LIN {X 0,Y 245.218,Z 452.069,A -85,B 0,C 180,E1 -20387.814,E2 -20387.814} C_VEL
LIN {X 0,Y 243.215,Z 463.262,A -85,B 0,C 180,E1 -20388.937,E2 -20388.937} C_VEL
LIN {X 0,Y 240.689,Z 473.992,A -85,B 0,C 180,E1 -20390.302,E2 -20390.302} C_VEL
LIN {X 0,Y 238.006,Z 484.022,A -85,B 0,C 180,E1 -20391.945,E2 -20391.945} C_VEL
LIN {X 0,Y 234.867,Z 493.616,A -85,B 0,C 180,E1 -20393.894,E2 -20393.894} C_VEL
LIN {X 0,Y 231.478,Z 503.094,A -85,B 0,C 180,E1 -20396.351,E2 -20396.351} C_VEL
LIN {X 0,Y 228.378,Z 510.879,A -85,B 0,C 180,E1 -20398.952,E2 -20398.952} C_VEL
LIN {X 0,Y 226.132,Z 516.237,A -85,B 0,C 180,E1 -20401.201,E2 -20401.201} C_VEL
LIN {X 0,Y 223.854,Z 521.339,A -85,B 0,C 180,E1 -20403.925,E2 -20403.925} C_VEL
LIN {X 0,Y 222.128,Z 525.113,A -85,B 0,C 180,E1 -20406.569,E2 -20406.569} C_VEL
LIN {X 0,Y 220.572,Z 528.106,A -85,B 0,C 180,E1 -20409.482,E2 -20409.482} C_VEL
LIN {X 0,Y 219.874,Z 529.432,A -85,B 0,C 180,E1 -20411.358,E2 -20411.358} C_VEL
LIN {X 0,Y 219.154,Z 530.646,A -85,B 0,C 180,E1 -20414.167,E2 -20414.167} C_VEL
LIN {X 0,Y 218.645,Z 530.949,A -85,B 0,C 180,E1 -20416.996,E2 -20416.996} C_VEL
LIN {X 0,Y 218.455,Z 529.925,A -85,B 0,C 180,E1 -20420.743,E2 -20420.743} C_VEL
LIN {X 0,Y 218.549,Z 528.815,A -85,B 0,C 180,E1 -20422.609,E2 -20422.609} C_VEL
LIN {X 0,Y 218.825,Z 527.086,A -85,B 0,C 180,E1 -20424.639,E2 -20424.639} C_VEL
LIN {X 0,Y 219.148,Z 524.142,A -85,B 0,C 180,E1 -20427.242,E2 -20427.242} C_VEL
LIN {X 0,Y 219.779,Z 519.981,A -85,B 0,C 180,E1 -20429.999,E2 -20429.999} C_VEL
LIN {X 0,Y 220.872,Z 513.649,A -85,B 0,C 180,E1 -20433.191,E2 -20433.191} C_VEL
LIN {X 0,Y 222.303,Z 506.749,A -85,B 0,C 180,E1 -20435.896,E2 -20435.896} C_VEL
LIN {X 0,Y 224.104,Z 498.102,A -85,B 0,C 180,E1 -20438.566,E2 -20438.566} C_VEL
LIN {X 0,Y 225.854,Z 489.254,A -85,B 0,C 180,E1 -20440.759,E2 -20440.759} C_VEL
LIN {X 0,Y 227.69,Z 479.531,A -85,B 0,C 180,E1 -20442.703,E2 -20442.703} C_VEL
LIN {X 0,Y 229.647,Z 468.829,A -85,B 0,C 180,E1 -20444.397,E2 -20444.397} C_VEL
LIN {X 0,Y 231.206,Z 458.803,A -85,B 0,C 180,E1 -20445.65,E2 -20445.65} C_VEL
LIN {X 0,Y 232.454,Z 445.756,A -85,B 0,C 180,E1 -20446.917,E2 -20446.917} C_VEL
LIN {X 0,Y 233.355,Z 433.916,A -85,B 0,C 180,E1 -20447.724,E2 -20447.724} C_VEL
LIN {X 0,Y 234.281,Z 421.059,A -85,B 0,C 180,E1 -20448.241,E2 -20448.241} C_VEL
LIN {X 0,Y 236.355,Z 359.149,A -85,B 0,C 180,E1 -20450.061,E2 -20450.061} C_VEL
LIN {X 0,Y 230.138,Z 342.133,A -85,B 0,C 180,E1 -20451.412,E2 -20451.412} C_VEL
LIN {X 0,Y 222.221,Z 326.344,A -85,B 0,C 180,E1 -20453.054,E2 -20453.054} C_VEL
LIN {X 0,Y 221.091,Z 324.032,A -85,B 0,C 180,E1 -20453.303,E2 -20453.303} C_VEL
LIN {X 0,Y 220.867,Z 322.97,A -85,B 0,C 180,E1 -20453.449,E2 -20453.449} C_VEL
LIN {X 0,Y 220.862,Z 322.967,A -85,B 0,C 180,E1 -20457.004,E2 -20457.004} C_VEL
LIN {X 0,Y 220.815,Z 322.977,A -85,B 0,C 180,E1 -20460.757,E2 -20460.757} C_VEL
LIN {X 0,Y 220.798,Z 322.981,A -85,B 0,C 180,E1 -20464.954,E2 -20464.954} C_VEL
LIN {X 0,Y 220.806,Z 322.976,A -85,B 0,C 180,E1 -20467.277,E2 -20467.277} C_VEL
LIN {X 0,Y 220.745,Z 322.985,A -85,B 0,C 180,E1 -20471.956,E2 -20471.956} C_VEL
LIN {X 0,Y 220.758,Z 322.98,A -85,B 0,C 180,E1 -20475.542,E2 -20475.542} C_VEL
LIN {X 0,Y 220.801,Z 322.97,A -85,B 0,C 180,E1 -20480.462,E2 -20480.462} C_VEL
LIN {X 0,Y 220.796,Z 322.98,A -85,B 0,C 180,E1 -20485.044,E2 -20485.044} C_VEL
LIN {X 0,Y 220.829,Z 322.961,A -85,B 0,C 180,E1 -20489.389,E2 -20489.389} C_VEL
LIN {X 0,Y 220.888,Z 322.969,A -85,B 0,C 180,E1 -20493.549,E2 -20493.549} C_VEL
LIN {X 0,Y 220.859,Z 322.965,A -85,B 0,C 180,E1 -20497.552,E2 -20497.552} C_VEL
LIN {X 0,Y 220.978,Z 322.955,A -85,B 0,C 180,E1 -20502.571,E2 -20502.571} C_VEL
LIN {X 0,Y 221.005,Z 322.951,A -85,B 0,C 180,E1 -20507.138,E2 -20507.138} C_VEL
LIN {X 0,Y 221.192,Z 322.915,A -85,B 0,C 180,E1 -20510.859,E2 -20510.859} C_VEL
LIN {X 0,Y 221.124,Z 322.941,A -85,B 0,C 180,E1 -20514.529,E2 -20514.529} C_VEL
LIN {X 0,Y 221.504,Z 322.885,A -85,B 0,C 180,E1 -20518.182,E2 -20518.182} C_VEL
LIN {X 0,Y 221.506,Z 322.877,A -85,B 0,C 180,E1 -20521.818,E2 -20521.818} C_VEL
LIN {X 0,Y 221.283,Z 322.917,A -85,B 0,C 180,E1 -20527.299,E2 -20527.299} C_VEL
LIN {X 0,Y 221.101,Z 322.925,A -85,B 0,C 180,E1 -20530.995,E2 -20530.995} C_VEL
LIN {X 0,Y 221.011,Z 322.956,A -85,B 0,C 180,E1 -20536.631,E2 -20536.631} C_VEL
LIN {X 0,Y 220.887,Z 322.971,A -85,B 0,C 180,E1 -20540.487,E2 -20540.487} C_VEL
LIN {X 0,Y 220.863,Z 322.974,A -85,B 0,C 180,E1 -20544.436,E2 -20544.436} C_VEL
LIN {X 0,Y 220.833,Z 322.978,A -85,B 0,C 180,E1 -20548.514,E2 -20548.514} C_VEL
LIN {X 0,Y 220.82,Z 322.981,A -85,B 0,C 180,E1 -20552.756,E2 -20552.756} C_VEL
LIN {X 0,Y 220.835,Z 322.979,A -85,B 0,C 180,E1 -20557.289,E2 -20557.289} C_VEL
LIN {X 0,Y 220.785,Z 322.98,A -85,B 0,C 180,E1 -20558.112,E2 -20558.112} C_VEL
LIN {X 0,Y 220.066,Z 323.075,A -85,B 0,C 180,E1 -20559.633,E2 -20559.633} C_VEL
LIN {X 0,Y 217.133,Z 323.441,A -85,B 0,C 180,E1 -20562.115,E2 -20562.115} C_VEL
LIN {X 0,Y 214.707,Z 323.742,A -85,B 0,C 180,E1 -20564.143,E2 -20564.143} C_VEL
LIN {X 0,Y 213.737,Z 323.864,A -85,B 0,C 180,E1 -20565.72,E2 -20565.72} C_VEL
LIN {X 0,Y 213.694,Z 323.867,A -85,B 0,C 180,E1 -20566.253,E2 -20566.253} C_VEL
LIN {X 0,Y 213.788,Z 324.003,A -85,B 0,C 180,E1 -20571.349,E2 -20571.349} C_VEL
LIN {X 0,Y 215.873,Z 332.818,A -85,B 0,C 180,E1 -20575.379,E2 -20575.379} C_VEL
LIN {X 0,Y 216.157,Z 334.104,A -85,B 0,C 180,E1 -20575.84,E2 -20575.84} C_VEL
LIN {X 0,Y 224.109,Z 353.666,A -85,B 0,C 180,E1 -20577.693,E2 -20577.693} C_VEL
LIN {X 0,Y 225.605,Z 358.401,A -85,B 0,C 180,E1 -20578.061,E2 -20578.061} C_VEL
LIN {X 0,Y 229.051,Z 388.519,A -85,B 0,C 180,E1 -20579.55,E2 -20579.55} C_VEL
LIN {X 0,Y 227.141,Z 442.514,A -85,B 0,C 180,E1 -20581.217,E2 -20581.217} C_VEL
LIN {X 0,Y 226.032,Z 455.896,A -85,B 0,C 180,E1 -20581.949,E2 -20581.949} C_VEL
LIN {X 0,Y 224.503,Z 468.707,A -85,B 0,C 180,E1 -20583.006,E2 -20583.006} C_VEL
LIN {X 0,Y 222.82,Z 480.076,A -85,B 0,C 180,E1 -20584.299,E2 -20584.299} C_VEL
LIN {X 0,Y 220.668,Z 491.795,A -85,B 0,C 180,E1 -20586.043,E2 -20586.043} C_VEL
LIN {X 0,Y 218.587,Z 502.341,A -85,B 0,C 180,E1 -20588.053,E2 -20588.053} C_VEL
LIN {X 0,Y 216.741,Z 511.35,A -85,B 0,C 180,E1 -20590.205,E2 -20590.205} C_VEL
LIN {X 0,Y 215.263,Z 518.901,A -85,B 0,C 180,E1 -20592.424,E2 -20592.424} C_VEL
LIN {X 0,Y 213.693,Z 526.627,A -85,B 0,C 180,E1 -20595.235,E2 -20595.235} C_VEL
LIN {X 0,Y 212.409,Z 533.745,A -85,B 0,C 180,E1 -20598.551,E2 -20598.551} C_VEL
LIN {X 0,Y 211.823,Z 538.462,A -85,B 0,C 180,E1 -20601.415,E2 -20601.415} C_VEL
LIN {X 0,Y 211.573,Z 542.044,A -85,B 0,C 180,E1 -20604.282,E2 -20604.282} C_VEL
LIN {X 0,Y 211.491,Z 543.863,A -85,B 0,C 180,E1 -20606.19,E2 -20606.19} C_VEL
LIN {X 0,Y 211.57,Z 545.225,A -85,B 0,C 180,E1 -20608.097,E2 -20608.097} C_VEL
LIN {X 0,Y 211.662,Z 546.184,A -85,B 0,C 180,E1 -20610.001,E2 -20610.001} C_VEL
LIN {X 0,Y 211.546,Z 546.738,A -85,B 0,C 180,E1 -20611.905,E2 -20611.905} C_VEL
LIN {X 0,Y 211.447,Z 546.827,A -85,B 0,C 180,E1 -20614.339,E2 -20614.339} C_VEL
LIN {X 0,Y 211.688,Z 545.948,A -85,B 0,C 180,E1 -20617.632,E2 -20617.632} C_VEL
LIN {X 0,Y 212.618,Z 543.469,A -85,B 0,C 180,E1 -20621.44,E2 -20621.44} C_VEL
LIN {X 0,Y 213.774,Z 540.493,A -85,B 0,C 180,E1 -20624.275,E2 -20624.275} C_VEL
LIN {X 0,Y 215.586,Z 536.498,A -85,B 0,C 180,E1 -20627.062,E2 -20627.062} C_VEL
LIN {X 0,Y 218.269,Z 530.392,A -85,B 0,C 180,E1 -20630.252,E2 -20630.252} C_VEL
LIN {X 0,Y 220.971,Z 523.75,A -85,B 0,C 180,E1 -20632.931,E2 -20632.931} C_VEL
LIN {X 0,Y 224.257,Z 515.533,A -85,B 0,C 180,E1 -20635.526,E2 -20635.526} C_VEL
LIN {X 0,Y 227.462,Z 507.142,A -85,B 0,C 180,E1 -20637.611,E2 -20637.611} C_VEL
LIN {X 0,Y 230.597,Z 497.976,A -85,B 0,C 180,E1 -20639.436,E2 -20639.436} C_VEL
LIN {X 0,Y 233.641,Z 488.025,A -85,B 0,C 180,E1 -20641.006,E2 -20641.006} C_VEL
LIN {X 0,Y 236.777,Z 475.482,A -85,B 0,C 180,E1 -20642.547,E2 -20642.547} C_VEL
LIN {X 0,Y 239.392,Z 463.039,A -85,B 0,C 180,E1 -20643.651,E2 -20643.651} C_VEL
LIN {X 0,Y 241.306,Z 449.921,A -85,B 0,C 180,E1 -20644.472,E2 -20644.472} C_VEL
LIN {X 0,Y 242.479,Z 436.547,A -85,B 0,C 180,E1 -20645.002,E2 -20645.002} C_VEL
LIN {X 0,Y 244.555,Z 394.353,A -85,B 0,C 180,E1 -20646.191,E2 -20646.191} C_VEL
LIN {X 0,Y 242.529,Z 381.265,A -85,B 0,C 180,E1 -20647.1,E2 -20647.1} C_VEL
LIN {X 0,Y 236.323,Z 367.487,A -85,B 0,C 180,E1 -20648.985,E2 -20648.985} C_VEL
LIN {X 0,Y 230.518,Z 355.918,A -85,B 0,C 180,E1 -20650.845,E2 -20650.845} C_VEL
LIN {X 0,Y 225.522,Z 347.08,A -85,B 0,C 180,E1 -20652.526,E2 -20652.526} C_VEL
LIN {X 0,Y 222.261,Z 341.762,A -85,B 0,C 180,E1 -20653.673,E2 -20653.673} C_VEL
LIN {X 0,Y 219.278,Z 336.956,A -85,B 0,C 180,E1 -20654.774,E2 -20654.774} C_VEL
LIN {X 0,Y 216.414,Z 332.444,A -85,B 0,C 180,E1 -20655.881,E2 -20655.881} C_VEL
LIN {X 0,Y 216.128,Z 331.625,A -85,B 0,C 180,E1 -20656.216,E2 -20656.216} C_VEL
LIN {X 0,Y 214.216,Z 325.551,A -85,B 0,C 180,E1 -20660.226,E2 -20660.226} C_VEL
LIN {X 0,Y 213.74,Z 323.86,A -85,B 0,C 180,E1 -20661.453,E2 -20661.453} C_VEL
LIN {X 0,Y 213.759,Z 323.848,A -85,B 0,C 180,E1 -20666.018,E2 -20666.018} C_VEL
LIN {X 0,Y 213.783,Z 323.849,A -85,B 0,C 180,E1 -20670.454,E2 -20670.454} C_VEL
LIN {X 0,Y 213.804,Z 323.851,A -85,B 0,C 180,E1 -20674.702,E2 -20674.702} C_VEL
LIN {X 0,Y 213.815,Z 323.85,A -85,B 0,C 180,E1 -20678.803,E2 -20678.803} C_VEL
LIN {X 0,Y 213.946,Z 323.831,A -85,B 0,C 180,E1 -20682.803,E2 -20682.803} C_VEL
LIN {X 0,Y 213.955,Z 323.824,A -85,B 0,C 180,E1 -20686.706,E2 -20686.706} C_VEL
LIN {X 0,Y 214.143,Z 323.795,A -85,B 0,C 180,E1 -20690.555,E2 -20690.555} C_VEL
LIN {X 0,Y 214.21,Z 323.796,A -85,B 0,C 180,E1 -20692.459,E2 -20692.459} C_VEL
LIN {X 0,Y 214.446,Z 323.756,A -85,B 0,C 180,E1 -20698.122,E2 -20698.122} C_VEL
LIN {X 0,Y 214.547,Z 323.745,A -85,B 0,C 180,E1 -20700,E2 -20700} C_VEL
LIN {X 0,Y 214.446,Z 323.764,A -85,B 0,C 180,E1 -20701.878,E2 -20701.878} C_VEL
LIN {X 0,Y 214.229,Z 323.785,A -85,B 0,C 180,E1 -20707.54,E2 -20707.54} C_VEL
LIN {X 0,Y 214.025,Z 323.816,A -85,B 0,C 180,E1 -20711.363,E2 -20711.363} C_VEL
LIN {X 0,Y 213.935,Z 323.833,A -85,B 0,C 180,E1 -20715.237,E2 -20715.237} C_VEL
LIN {X 0,Y 213.838,Z 323.847,A -85,B 0,C 180,E1 -20719.187,E2 -20719.187} C_VEL
LIN {X 0,Y 213.812,Z 323.849,A -85,B 0,C 180,E1 -20723.231,E2 -20723.231} C_VEL
LIN {X 0,Y 213.83,Z 323.84,A -85,B 0,C 180,E1 -20727.449,E2 -20727.449} C_VEL
LIN {X 0,Y 213.767,Z 323.851,A -85,B 0,C 180,E1 -20732.852,E2 -20732.852} C_VEL
LIN {X 0,Y 213.756,Z 323.856,A -85,B 0,C 180,E1 -20733.346,E2 -20733.346} C_VEL
LIN {X 0,Y 214.688,Z 326.586,A -85,B 0,C 180,E1 -20733.814,E2 -20733.814} C_VEL
LIN {X 0,Y 216.886,Z 328.881,A -85,B 0,C 180,E1 -20734.64,E2 -20734.64} C_VEL
LIN {X 0,Y 217.628,Z 329.93,A -85,B 0,C 180,E1 -20734.926,E2 -20734.926} C_VEL
LIN {X 0,Y 219.934,Z 333.195,A -85,B 0,C 180,E1 -20735.792,E2 -20735.792} C_VEL
LIN {X 0,Y 221.203,Z 334.982,A -85,B 0,C 180,E1 -20736.253,E2 -20736.253} C_VEL
LIN {X 0,Y 224.639,Z 339.803,A -85,B 0,C 180,E1 -20737.453,E2 -20737.453} C_VEL
LIN {X 0,Y 229.579,Z 346.935,A -85,B 0,C 180,E1 -20739.081,E2 -20739.081} C_VEL
LIN {X 0,Y 235.077,Z 355.949,A -85,B 0,C 180,E1 -20740.807,E2 -20740.807} C_VEL
LIN {X 0,Y 242.231,Z 369.906,A -85,B 0,C 180,E1 -20742.95,E2 -20742.95} C_VEL
LIN {X 0,Y 245.346,Z 376.787,A -85,B 0,C 180,E1 -20743.854,E2 -20743.854} C_VEL
LIN {X 0,Y 242.644,Z 428.181,A -85,B 0,C 180,E1 -20745.321,E2 -20745.321} C_VEL
LIN {X 0,Y 241.226,Z 441.469,A -85,B 0,C 180,E1 -20745.998,E2 -20745.998} C_VEL
LIN {X 0,Y 239.694,Z 451.476,A -85,B 0,C 180,E1 -20746.735,E2 -20746.735} C_VEL
LIN {X 0,Y 237.49,Z 463.347,A -85,B 0,C 180,E1 -20747.929,E2 -20747.929} C_VEL
LIN {X 0,Y 234.756,Z 474.507,A -85,B 0,C 180,E1 -20749.372,E2 -20749.372} C_VEL
LIN {X 0,Y 231.96,Z 484.478,A -85,B 0,C 180,E1 -20751.046,E2 -20751.046} C_VEL
LIN {X 0,Y 228.684,Z 494.062,A -85,B 0,C 180,E1 -20753.038,E2 -20753.038} C_VEL
LIN {X 0,Y 225.431,Z 502.734,A -85,B 0,C 180,E1 -20755.322,E2 -20755.322} C_VEL
LIN {X 0,Y 222.628,Z 509.492,A -85,B 0,C 180,E1 -20757.543,E2 -20757.543} C_VEL
LIN {X 0,Y 219.746,Z 516.103,A -85,B 0,C 180,E1 -20760.282,E2 -20760.282} C_VEL
LIN {X 0,Y 217.292,Z 521.306,A -85,B 0,C 180,E1 -20763.075,E2 -20763.075} C_VEL
LIN {X 0,Y 215.26,Z 525.486,A -85,B 0,C 180,E1 -20766.088,E2 -20766.088} C_VEL
LIN {X 0,Y 213.769,Z 528.221,A -85,B 0,C 180,E1 -20768.798,E2 -20768.798} C_VEL
LIN {X 0,Y 212.968,Z 529.584,A -85,B 0,C 180,E1 -20770.73,E2 -20770.73} C_VEL
LIN {X 0,Y 211.966,Z 531.099,A -85,B 0,C 180,E1 -20774.617,E2 -20774.617} C_VEL
LIN {X 0,Y 211.626,Z 531.234,A -85,B 0,C 180,E1 -20776.557,E2 -20776.557} C_VEL
LIN {X 0,Y 211.369,Z 530.276,A -85,B 0,C 180,E1 -20780.429,E2 -20780.429} C_VEL
LIN {X 0,Y 211.426,Z 529.214,A -85,B 0,C 180,E1 -20782.358,E2 -20782.358} C_VEL
LIN {X 0,Y 211.748,Z 527.318,A -85,B 0,C 180,E1 -20784.69,E2 -20784.69} C_VEL
LIN {X 0,Y 212.164,Z 523.421,A -85,B 0,C 180,E1 -20788.101,E2 -20788.101} C_VEL
LIN {X 0,Y 212.967,Z 518.963,A -85,B 0,C 180,E1 -20790.944,E2 -20790.944} C_VEL
LIN {X 0,Y 214.219,Z 512.224,A -85,B 0,C 180,E1 -20794.232,E2 -20794.232} C_VEL
LIN {X 0,Y 215.839,Z 504.882,A -85,B 0,C 180,E1 -20797.013,E2 -20797.013} C_VEL
LIN {X 0,Y 217.768,Z 495.778,A -85,B 0,C 180,E1 -20799.754,E2 -20799.754} C_VEL
LIN {X 0,Y 219.979,Z 485.237,A -85,B 0,C 180,E1 -20802.218,E2 -20802.218} C_VEL
LIN {X 0,Y 222.003,Z 474.515,A -85,B 0,C 180,E1 -20804.201,E2 -20804.201} C_VEL
LIN {X 0,Y 224.002,Z 464.022,A -85,B 0,C 180,E1 -20805.699,E2 -20805.699} C_VEL
LIN {X 0,Y 225.416,Z 451.564,A -85,B 0,C 180,E1 -20807.111,E2 -20807.111} C_VEL
LIN {X 0,Y 226.502,Z 438.518,A -85,B 0,C 180,E1 -20808.186,E2 -20808.186} C_VEL
LIN {X 0,Y 227.505,Z 425.949,A -85,B 0,C 180,E1 -20808.82,E2 -20808.82} C_VEL
LIN {X 0,Y 230.008,Z 361.903,A -85,B 0,C 180,E1 -20810.746,E2 -20810.746} C_VEL
LIN {X 0,Y 229.55,Z 359.483,A -85,B 0,C 180,E1 -20810.888,E2 -20810.888} C_VEL
LIN {X 0,Y 223.85,Z 344.115,A -85,B 0,C 180,E1 -20812.183,E2 -20812.183} C_VEL
LIN {X 0,Y 216.303,Z 329.378,A -85,B 0,C 180,E1 -20813.818,E2 -20813.818} C_VEL
LIN {X 0,Y 214.031,Z 324.886,A -85,B 0,C 180,E1 -20814.339,E2 -20814.339} C_VEL
LIN {X 0,Y 213.799,Z 323.851,A -85,B 0,C 180,E1 -20814.45,E2 -20814.45} C_VEL
LIN {X 0,Y 213.784,Z 323.851,A -85,B 0,C 180,E1 -20817.427,E2 -20817.427} C_VEL
LIN {X 0,Y 213.756,Z 323.856,A -85,B 0,C 180,E1 -20821.738,E2 -20821.738} C_VEL
LIN {X 0,Y 213.74,Z 323.86,A -85,B 0,C 180,E1 -20826.287,E2 -20826.287} C_VEL
LIN {X 0,Y 213.694,Z 323.867,A -85,B 0,C 180,E1 -20831.127,E2 -20831.127} C_VEL
LIN {X 0,Y 213.697,Z 323.854,A -85,B 0,C 180,E1 -20833.679,E2 -20833.679} C_VEL
LIN {X 0,Y 213.698,Z 323.861,A -85,B 0,C 180,E1 -20836.344,E2 -20836.344} C_VEL
LIN {X 0,Y 213.711,Z 323.858,A -85,B 0,C 180,E1 -20839.142,E2 -20839.142} C_VEL
LIN {X 0,Y 213.739,Z 323.856,A -85,B 0,C 180,E1 -20843.711,E2 -20843.711} C_VEL
LIN {X 0,Y 213.775,Z 323.843,A -85,B 0,C 180,E1 -20848.731,E2 -20848.731} C_VEL
LIN {X 0,Y 213.821,Z 323.845,A -85,B 0,C 180,E1 -20852.603,E2 -20852.603} C_VEL
LIN {X 0,Y 213.813,Z 323.847,A -85,B 0,C 180,E1 -20856.973,E2 -20856.973} C_VEL
LIN {X 0,Y 213.938,Z 323.831,A -85,B 0,C 180,E1 -20862.803,E2 -20862.803} C_VEL
LIN {X 0,Y 213.947,Z 323.83,A -85,B 0,C 180,E1 -20866.706,E2 -20866.706} C_VEL
LIN {X 0,Y 214.13,Z 323.792,A -85,B 0,C 180,E1 -20870.555,E2 -20870.555} C_VEL
LIN {X 0,Y 214.085,Z 323.818,A -85,B 0,C 180,E1 -20874.348,E2 -20874.348} C_VEL
LIN {X 0,Y 214.437,Z 323.765,A -85,B 0,C 180,E1 -20878.122,E2 -20878.122} C_VEL
LIN {X 0,Y 214.54,Z 323.742,A -85,B 0,C 180,E1 -20880,E2 -20880} C_VEL
LIN {X 0,Y 214.439,Z 323.757,A -85,B 0,C 180,E1 -20881.878,E2 -20881.878} C_VEL
LIN {X 0,Y 214.221,Z 323.797,A -85,B 0,C 180,E1 -20887.541,E2 -20887.541} C_VEL
LIN {X 0,Y 214.017,Z 323.807,A -85,B 0,C 180,E1 -20891.364,E2 -20891.364} C_VEL
LIN {X 0,Y 213.927,Z 323.837,A -85,B 0,C 180,E1 -20895.238,E2 -20895.238} C_VEL
LIN {X 0,Y 213.835,Z 323.849,A -85,B 0,C 180,E1 -20899.188,E2 -20899.188} C_VEL
LIN {X 0,Y 213.843,Z 323.849,A -85,B 0,C 180,E1 -20903.228,E2 -20903.228} C_VEL
LIN {X 0,Y 213.825,Z 323.852,A -85,B 0,C 180,E1 -20907.451,E2 -20907.451} C_VEL
LIN {X 0,Y 213.775,Z 323.858,A -85,B 0,C 180,E1 -20911.737,E2 -20911.737} C_VEL
LIN {X 0,Y 213.749,Z 323.86,A -85,B 0,C 180,E1 -20916.288,E2 -20916.288} C_VEL
LIN {X 0,Y 213.711,Z 323.868,A -85,B 0,C 180,E1 -20921.126,E2 -20921.126} C_VEL
LIN {X 0,Y 213.7,Z 323.87,A -85,B 0,C 180,E1 -20923.681,E2 -20923.681} C_VEL
LIN {X 0,Y 213.694,Z 323.867,A -85,B 0,C 180,E1 -20926.253,E2 -20926.253} C_VEL
LIN {X 0,Y 213.062,Z 323.958,A -85,B 0,C 180,E1 -20927.331,E2 -20927.331} C_VEL
LIN {X 0,Y 210.239,Z 324.297,A -85,B 0,C 180,E1 -20929.033,E2 -20929.033} C_VEL
LIN {X 0,Y 208.019,Z 325.277,A -85,B 0,C 180,E1 -20930.371,E2 -20930.371} C_VEL
LIN {X 0,Y 207.272,Z 326.653,A -85,B 0,C 180,E1 -20931.382,E2 -20931.382} C_VEL
LIN {X 0,Y 207.337,Z 327.264,A -85,B 0,C 180,E1 -20931.707,E2 -20931.707} C_VEL
LIN {X 0,Y 208.832,Z 333.629,A -85,B 0,C 180,E1 -20934.669,E2 -20934.669} C_VEL
LIN {X 0,Y 217.546,Z 354.665,A -85,B 0,C 180,E1 -20936.813,E2 -20936.813} C_VEL
LIN {X 0,Y 219.489,Z 360.434,A -85,B 0,C 180,E1 -20937.302,E2 -20937.302} C_VEL
LIN {X 0,Y 222.721,Z 390.003,A -85,B 0,C 180,E1 -20938.803,E2 -20938.803} C_VEL
LIN {X 0,Y 220.662,Z 443.037,A -85,B 0,C 180,E1 -20940.485,E2 -20940.485} C_VEL
LIN {X 0,Y 219.409,Z 456.917,A -85,B 0,C 180,E1 -20941.285,E2 -20941.285} C_VEL
LIN {X 0,Y 217.861,Z 469.364,A -85,B 0,C 180,E1 -20942.374,E2 -20942.374} C_VEL
LIN {X 0,Y 215.803,Z 482.075,A -85,B 0,C 180,E1 -20943.92,E2 -20943.92} C_VEL
LIN {X 0,Y 213.648,Z 493.386,A -85,B 0,C 180,E1 -20945.722,E2 -20945.722} C_VEL
LIN {X 0,Y 211.551,Z 503.552,A -85,B 0,C 180,E1 -20947.798,E2 -20947.798} C_VEL
LIN {X 0,Y 209.445,Z 513.561,A -85,B 0,C 180,E1 -20950.395,E2 -20950.395} C_VEL
LIN {X 0,Y 207.606,Z 522.353,A -85,B 0,C 180,E1 -20953.278,E2 -20953.278} C_VEL
LIN {X 0,Y 206.061,Z 529.336,A -85,B 0,C 180,E1 -20956.189,E2 -20956.189} C_VEL
LIN {X 0,Y 205.148,Z 534.934,A -85,B 0,C 180,E1 -20959.141,E2 -20959.141} C_VEL
LIN {X 0,Y 204.63,Z 539.314,A -85,B 0,C 180,E1 -20962.105,E2 -20962.105} C_VEL
LIN {X 0,Y 204.412,Z 543.092,A -85,B 0,C 180,E1 -20965.614,E2 -20965.614} C_VEL
LIN {X 0,Y 204.466,Z 544.879,A -85,B 0,C 180,E1 -20968.031,E2 -20968.031} C_VEL
LIN {X 0,Y 204.575,Z 545.862,A -85,B 0,C 180,E1 -20970.001,E2 -20970.001} C_VEL
LIN {X 0,Y 204.46,Z 546.438,A -85,B 0,C 180,E1 -20971.971,E2 -20971.971} C_VEL
LIN {X 0,Y 204.348,Z 546.606,A -85,B 0,C 180,E1 -20974.145,E2 -20974.145} C_VEL
LIN {X 0,Y 204.64,Z 545.74,A -85,B 0,C 180,E1 -20977.897,E2 -20977.897} C_VEL
LIN {X 0,Y 205.619,Z 543.319,A -85,B 0,C 180,E1 -20981.835,E2 -20981.835} C_VEL
LIN {X 0,Y 206.881,Z 540.383,A -85,B 0,C 180,E1 -20984.762,E2 -20984.762} C_VEL
LIN {X 0,Y 208.801,Z 536.439,A -85,B 0,C 180,E1 -20987.634,E2 -20987.634} C_VEL
LIN {X 0,Y 211.158,Z 531.385,A -85,B 0,C 180,E1 -20990.456,E2 -20990.456} C_VEL
LIN {X 0,Y 213.911,Z 525.065,A -85,B 0,C 180,E1 -20993.22,E2 -20993.22} C_VEL
LIN {X 0,Y 217.252,Z 517.184,A -85,B 0,C 180,E1 -20995.895,E2 -20995.895} C_VEL
LIN {X 0,Y 221.208,Z 507.399,A -85,B 0,C 180,E1 -20998.462,E2 -20998.462} C_VEL
LIN {X 0,Y 224.462,Z 498.365,A -85,B 0,C 180,E1 -21000.324,E2 -21000.324} C_VEL
LIN {X 0,Y 228.015,Z 487.182,A -85,B 0,C 180,E1 -21002.12,E2 -21002.12} C_VEL
LIN {X 0,Y 230.863,Z 476.261,A -85,B 0,C 180,E1 -21003.489,E2 -21003.489} C_VEL
LIN {X 0,Y 233.567,Z 464.171,A -85,B 0,C 180,E1 -21004.608,E2 -21004.608} C_VEL
LIN {X 0,Y 235.601,Z 451.361,A -85,B 0,C 180,E1 -21005.462,E2 -21005.462} C_VEL
LIN {X 0,Y 236.908,Z 437.774,A -85,B 0,C 180,E1 -21006.041,E2 -21006.041} C_VEL
LIN {X 0,Y 239.115,Z 395.539,A -85,B 0,C 180,E1 -21007.253,E2 -21007.253} C_VEL
LIN {X 0,Y 237.536,Z 384.595,A -85,B 0,C 180,E1 -21008.024,E2 -21008.024} C_VEL
LIN {X 0,Y 230.881,Z 369.544,A -85,B 0,C 180,E1 -21010.169,E2 -21010.169} C_VEL
LIN {X 0,Y 224.679,Z 357.345,A -85,B 0,C 180,E1 -21012.284,E2 -21012.284} C_VEL
LIN {X 0,Y 218.487,Z 346.829,A -85,B 0,C 180,E1 -21014.526,E2 -21014.526} C_VEL
LIN {X 0,Y 215.531,Z 342.013,A -85,B 0,C 180,E1 -21015.673,E2 -21015.673} C_VEL
LIN {X 0,Y 212.12,Z 336.781,A -85,B 0,C 180,E1 -21017.056,E2 -21017.056} C_VEL
LIN {X 0,Y 209.174,Z 332.353,A -85,B 0,C 180,E1 -21018.319,E2 -21018.319} C_VEL
LIN {X 0,Y 208.756,Z 331.386,A -85,B 0,C 180,E1 -21018.631,E2 -21018.631} C_VEL
LIN {X 0,Y 207.706,Z 327.876,A -85,B 0,C 180,E1 -21021.1,E2 -21021.1} C_VEL
LIN {X 0,Y 206.701,Z 324.731,A -85,B 0,C 180,E1 -21023.637,E2 -21023.637} C_VEL
LIN {X 0,Y 206.728,Z 324.731,A -85,B 0,C 180,E1 -21028.202,E2 -21028.202} C_VEL
LIN {X 0,Y 206.769,Z 324.725,A -85,B 0,C 180,E1 -21032.096,E2 -21032.096} C_VEL
LIN {X 0,Y 206.788,Z 324.718,A -85,B 0,C 180,E1 -21036.584,E2 -21036.584} C_VEL
LIN {X 0,Y 206.875,Z 324.706,A -85,B 0,C 180,E1 -21042.196,E2 -21042.196} C_VEL
LIN {X 0,Y 206.897,Z 324.7,A -85,B 0,C 180,E1 -21046.244,E2 -21046.244} C_VEL
LIN {X 0,Y 207.101,Z 324.671,A -85,B 0,C 180,E1 -21050.231,E2 -21050.231} C_VEL
LIN {X 0,Y 207.066,Z 324.674,A -85,B 0,C 180,E1 -21054.156,E2 -21054.156} C_VEL
LIN {X 0,Y 207.383,Z 324.636,A -85,B 0,C 180,E1 -21058.058,E2 -21058.058} C_VEL
LIN {X 0,Y 207.513,Z 324.621,A -85,B 0,C 180,E1 -21060,E2 -21060} C_VEL
LIN {X 0,Y 207.382,Z 324.643,A -85,B 0,C 180,E1 -21061.942,E2 -21061.942} C_VEL
LIN {X 0,Y 207.169,Z 324.663,A -85,B 0,C 180,E1 -21067.799,E2 -21067.799} C_VEL
LIN {X 0,Y 206.945,Z 324.695,A -85,B 0,C 180,E1 -21071.757,E2 -21071.757} C_VEL
LIN {X 0,Y 206.868,Z 324.708,A -85,B 0,C 180,E1 -21075.77,E2 -21075.77} C_VEL
LIN {X 0,Y 206.764,Z 324.722,A -85,B 0,C 180,E1 -21079.871,E2 -21079.871} C_VEL
LIN {X 0,Y 206.748,Z 324.722,A -85,B 0,C 180,E1 -21084.074,E2 -21084.074} C_VEL
LIN {X 0,Y 206.738,Z 324.72,A -85,B 0,C 180,E1 -21088.419,E2 -21088.419} C_VEL
LIN {X 0,Y 206.722,Z 324.732,A -85,B 0,C 180,E1 -21090.9,E2 -21090.9} C_VEL
LIN {X 0,Y 207.563,Z 327.231,A -85,B 0,C 180,E1 -21091.36,E2 -21091.36} C_VEL
LIN {X 0,Y 209.337,Z 329.401,A -85,B 0,C 180,E1 -21092.13,E2 -21092.13} C_VEL
LIN {X 0,Y 210.463,Z 330.303,A -85,B 0,C 180,E1 -21092.579,E2 -21092.579} C_VEL
LIN {X 0,Y 212.448,Z 333.539,A -85,B 0,C 180,E1 -21093.436,E2 -21093.436} C_VEL
LIN {X 0,Y 214.203,Z 335.41,A -85,B 0,C 180,E1 -21094.116,E2 -21094.116} C_VEL
LIN {X 0,Y 216.867,Z 339.123,A -85,B 0,C 180,E1 -21095.152,E2 -21095.152} C_VEL
LIN {X 0,Y 225.448,Z 351.594,A -85,B 0,C 180,E1 -21098.214,E2 -21098.214} C_VEL
LIN {X 0,Y 230.848,Z 360.543,A -85,B 0,C 180,E1 -21099.99,E2 -21099.99} C_VEL
LIN {X 0,Y 237.522,Z 373.867,A -85,B 0,C 180,E1 -21102.096,E2 -21102.096} C_VEL
LIN {X 0,Y 239.888,Z 379.125,A -85,B 0,C 180,E1 -21102.817,E2 -21102.817} C_VEL
LIN {X 0,Y 237.104,Z 429.221,A -85,B 0,C 180,E1 -21104.279,E2 -21104.279} C_VEL
LIN {X 0,Y 235.5,Z 443.104,A -85,B 0,C 180,E1 -21105.016,E2 -21105.016} C_VEL
LIN {X 0,Y 233.823,Z 453.34,A -85,B 0,C 180,E1 -21105.817,E2 -21105.817} C_VEL
LIN {X 0,Y 231.68,Z 464.189,A -85,B 0,C 180,E1 -21106.954,E2 -21106.954} C_VEL
LIN {X 0,Y 228.897,Z 475.035,A -85,B 0,C 180,E1 -21108.396,E2 -21108.396} C_VEL
LIN {X 0,Y 225.62,Z 486.044,A -85,B 0,C 180,E1 -21110.314,E2 -21110.314} C_VEL
LIN {X 0,Y 222.11,Z 495.724,A -85,B 0,C 180,E1 -21112.427,E2 -21112.427} C_VEL
LIN {X 0,Y 218.866,Z 503.892,A -85,B 0,C 180,E1 -21114.69,E2 -21114.69} C_VEL
LIN {X 0,Y 215.447,Z 511.655,A -85,B 0,C 180,E1 -21117.435,E2 -21117.435} C_VEL
LIN {X 0,Y 212.505,Z 517.845,A -85,B 0,C 180,E1 -21120.258,E2 -21120.258} C_VEL
LIN {X 0,Y 210.058,Z 522.716,A -85,B 0,C 180,E1 -21123.148,E2 -21123.148} C_VEL
LIN {X 0,Y 208.104,Z 526.42,A -85,B 0,C 180,E1 -21126.092,E2 -21126.092} C_VEL
LIN {X 0,Y 207.008,Z 528.317,A -85,B 0,C 180,E1 -21128.07,E2 -21128.07} C_VEL
LIN {X 0,Y 206.111,Z 529.736,A -85,B 0,C 180,E1 -21130.063,E2 -21130.063} C_VEL
LIN {X 0,Y 204.97,Z 531.318,A -85,B 0,C 180,E1 -21134.079,E2 -21134.079} C_VEL
LIN {X 0,Y 204.589,Z 531.514,A -85,B 0,C 180,E1 -21136.085,E2 -21136.085} C_VEL
LIN {X 0,Y 204.259,Z 530.628,A -85,B 0,C 180,E1 -21140.093,E2 -21140.093} C_VEL
LIN {X 0,Y 204.331,Z 529.598,A -85,B 0,C 180,E1 -21142.091,E2 -21142.091} C_VEL
LIN {X 0,Y 204.658,Z 527.513,A -85,B 0,C 180,E1 -21144.786,E2 -21144.786} C_VEL
LIN {X 0,Y 205.074,Z 523.94,A -85,B 0,C 180,E1 -21148.035,E2 -21148.035} C_VEL
LIN {X 0,Y 205.872,Z 519.558,A -85,B 0,C 180,E1 -21150.977,E2 -21150.977} C_VEL
LIN {X 0,Y 206.952,Z 513.997,A -85,B 0,C 180,E1 -21153.893,E2 -21153.893} C_VEL
LIN {X 0,Y 208.507,Z 507.049,A -85,B 0,C 180,E1 -21156.774,E2 -21156.774} C_VEL
LIN {X 0,Y 210.464,Z 498.343,A -85,B 0,C 180,E1 -21159.61,E2 -21159.61} C_VEL
LIN {X 0,Y 212.386,Z 489.438,A -85,B 0,C 180,E1 -21161.935,E2 -21161.935} C_VEL
LIN {X 0,Y 214.408,Z 479.641,A -85,B 0,C 180,E1 -21163.988,E2 -21163.988} C_VEL
LIN {X 0,Y 216.524,Z 468.8,A -85,B 0,C 180,E1 -21165.772,E2 -21165.772} C_VEL
LIN {X 0,Y 218.188,Z 458.638,A -85,B 0,C 180,E1 -21167.092,E2 -21167.092} C_VEL
LIN {X 0,Y 219.439,Z 446.657,A -85,B 0,C 180,E1 -21168.315,E2 -21168.315} C_VEL
LIN {X 0,Y 220.377,Z 435.411,A -85,B 0,C 180,E1 -21169.139,E2 -21169.139} C_VEL
LIN {X 0,Y 221.33,Z 422.431,A -85,B 0,C 180,E1 -21169.716,E2 -21169.716} C_VEL
LIN {X 0,Y 223.577,Z 362.258,A -85,B 0,C 180,E1 -21171.571,E2 -21171.571} C_VEL
LIN {X 0,Y 218.256,Z 347.659,A -85,B 0,C 180,E1 -21172.845,E2 -21172.845} C_VEL
LIN {X 0,Y 210.088,Z 331.592,A -85,B 0,C 180,E1 -21174.707,E2 -21174.707} C_VEL
LIN {X 0,Y 207.001,Z 325.992,A -85,B 0,C 180,E1 -21175.439,E2 -21175.439} C_VEL
LIN {X 0,Y 206.742,Z 324.728,A -85,B 0,C 180,E1 -21175.566,E2 -21175.566} C_VEL
LIN {X 0,Y 206.693,Z 324.735,A -85,B 0,C 180,E1 -21180.664,E2 -21180.664} C_VEL
LIN {X 0,Y 206.696,Z 324.739,A -85,B 0,C 180,E1 -21185.31,E2 -21185.31} C_VEL
LIN {X 0,Y 206.643,Z 324.742,A -85,B 0,C 180,E1 -21190.253,E2 -21190.253} C_VEL
LIN {X 0,Y 206.625,Z 324.733,A -85,B 0,C 180,E1 -21194.416,E2 -21194.416} C_VEL
LIN {X 0,Y 206.636,Z 324.742,A -85,B 0,C 180,E1 -21198.437,E2 -21198.437} C_VEL
LIN {X 0,Y 206.674,Z 324.727,A -85,B 0,C 180,E1 -21202.259,E2 -21202.259} C_VEL
LIN {X 0,Y 206.694,Z 324.734,A -85,B 0,C 180,E1 -21207.042,E2 -21207.042} C_VEL
LIN {X 0,Y 206.759,Z 324.722,A -85,B 0,C 180,E1 -21212.097,E2 -21212.097} C_VEL
LIN {X 0,Y 206.748,Z 324.727,A -85,B 0,C 180,E1 -21216.604,E2 -21216.604} C_VEL
LIN {X 0,Y 206.867,Z 324.709,A -85,B 0,C 180,E1 -21222.196,E2 -21222.196} C_VEL
LIN {X 0,Y 206.889,Z 324.711,A -85,B 0,C 180,E1 -21226.244,E2 -21226.244} C_VEL
LIN {X 0,Y 207.074,Z 324.669,A -85,B 0,C 180,E1 -21230.23,E2 -21230.23} C_VEL
LIN {X 0,Y 207.047,Z 324.693,A -85,B 0,C 180,E1 -21234.156,E2 -21234.156} C_VEL
LIN {X 0,Y 207.374,Z 324.645,A -85,B 0,C 180,E1 -21238.058,E2 -21238.058} C_VEL
LIN {X 0,Y 207.505,Z 324.617,A -85,B 0,C 180,E1 -21240,E2 -21240} C_VEL
LIN {X 0,Y 207.376,Z 324.636,A -85,B 0,C 180,E1 -21241.942,E2 -21241.942} C_VEL
LIN {X 0,Y 207.161,Z 324.677,A -85,B 0,C 180,E1 -21247.799,E2 -21247.799} C_VEL
LIN {X 0,Y 206.937,Z 324.69,A -85,B 0,C 180,E1 -21251.758,E2 -21251.758} C_VEL
LIN {X 0,Y 206.861,Z 324.716,A -85,B 0,C 180,E1 -21255.771,E2 -21255.771} C_VEL
LIN {X 0,Y 206.779,Z 324.727,A -85,B 0,C 180,E1 -21259.87,E2 -21259.87} C_VEL
LIN {X 0,Y 206.759,Z 324.73,A -85,B 0,C 180,E1 -21264.073,E2 -21264.073} C_VEL
LIN {X 0,Y 206.74,Z 324.734,A -85,B 0,C 180,E1 -21268.42,E2 -21268.42} C_VEL
LIN {X 0,Y 206.705,Z 324.739,A -85,B 0,C 180,E1 -21272.957,E2 -21272.957} C_VEL
LIN {X 0,Y 206.718,Z 324.74,A -85,B 0,C 180,E1 -21275.321,E2 -21275.321} C_VEL
LIN {X 0,Y 206.662,Z 324.744,A -85,B 0,C 180,E1 -21280.251,E2 -21280.251} C_VEL
LIN {X 0,Y 206.628,Z 324.749,A -85,B 0,C 180,E1 -21285.584,E2 -21285.584} C_VEL
LIN {X 0,Y 206.761,Z 324.885,A -85,B 0,C 180,E1 -21290.543,E2 -21290.543} C_VEL
LIN {X 0,Y 207.337,Z 327.264,A -85,B 0,C 180,E1 -21291.707,E2 -21291.707} C_VEL
LIN {X 0,Y 207.694,Z 329.601,A -85,B 0,C 180,E1 -21292.557,E2 -21292.557} C_VEL
LIN {X 0,Y 207.894,Z 334.219,A -85,B 0,C 180,E1 -21293.559,E2 -21293.559} C_VEL
LIN {X 0,Y 207.985,Z 339.539,A -85,B 0,C 180,E1 -21294.296,E2 -21294.296} C_VEL
LIN {X 0,Y 208.563,Z 347.244,A -85,B 0,C 180,E1 -21295.06,E2 -21295.06} C_VEL
LIN {X 0,Y 209.902,Z 352.888,A -85,B 0,C 180,E1 -21295.589,E2 -21295.589} C_VEL
LIN {X 0,Y 210.618,Z 354.668,A -85,B 0,C 180,E1 -21295.775,E2 -21295.775} C_VEL
LIN {X 0,Y 213.387,Z 362.474,A -85,B 0,C 180,E1 -21296.496,E2 -21296.496} C_VEL
LIN {X 0,Y 216.373,Z 391.44,A -85,B 0,C 180,E1 -21298.006,E2 -21298.006} C_VEL
LIN {X 0,Y 214.326,Z 442.22,A -85,B 0,C 180,E1 -21299.647,E2 -21299.647} C_VEL
LIN {X 0,Y 213.116,Z 455.647,A -85,B 0,C 180,E1 -21300.422,E2 -21300.422} C_VEL
LIN {X 0,Y 211.587,Z 467.826,A -85,B 0,C 180,E1 -21301.481,E2 -21301.481} C_VEL
LIN {X 0,Y 209.751,Z 479.293,A -85,B 0,C 180,E1 -21302.838,E2 -21302.838} C_VEL
LIN {X 0,Y 207.337,Z 491.049,A -85,B 0,C 180,E1 -21304.664,E2 -21304.664} C_VEL
LIN {X 0,Y 205.172,Z 501.645,A -85,B 0,C 180,E1 -21306.803,E2 -21306.803} C_VEL
LIN {X 0,Y 202.906,Z 511.686,A -85,B 0,C 180,E1 -21309.374,E2 -21309.374} C_VEL
LIN {X 0,Y 201.344,Z 518.963,A -85,B 0,C 180,E1 -21311.692,E2 -21311.692} C_VEL
LIN {X 0,Y 199.648,Z 526.575,A -85,B 0,C 180,E1 -21314.693,E2 -21314.693} C_VEL
LIN {X 0,Y 198.439,Z 532.687,A -85,B 0,C 180,E1 -21317.732,E2 -21317.732} C_VEL
LIN {X 0,Y 197.722,Z 537.516,A -85,B 0,C 180,E1 -21320.797,E2 -21320.797} C_VEL
LIN {X 0,Y 197.408,Z 541.205,A -85,B 0,C 180,E1 -21323.87,E2 -21323.87} C_VEL
LIN {X 0,Y 197.326,Z 543.102,A -85,B 0,C 180,E1 -21325.916,E2 -21325.916} C_VEL
LIN {X 0,Y 197.366,Z 544.533,A -85,B 0,C 180,E1 -21327.96,E2 -21327.96} C_VEL
LIN {X 0,Y 197.49,Z 545.539,A -85,B 0,C 180,E1 -21330.001,E2 -21330.001} C_VEL
LIN {X 0,Y 197.357,Z 546.138,A -85,B 0,C 180,E1 -21332.042,E2 -21332.042} C_VEL
LIN {X 0,Y 197.252,Z 546.348,A -85,B 0,C 180,E1 -21334.087,E2 -21334.087} C_VEL
LIN {X 0,Y 197.344,Z 546.142,A -85,B 0,C 180,E1 -21336.134,E2 -21336.134} C_VEL
LIN {X 0,Y 198.028,Z 544.54,A -85,B 0,C 180,E1 -21340.222,E2 -21340.222} C_VEL
LIN {X 0,Y 198.638,Z 543.16,A -85,B 0,C 180,E1 -21342.257,E2 -21342.257} C_VEL
LIN {X 0,Y 200.012,Z 540.272,A -85,B 0,C 180,E1 -21345.281,E2 -21345.281} C_VEL
LIN {X 0,Y 202.041,Z 536.382,A -85,B 0,C 180,E1 -21348.245,E2 -21348.245} C_VEL
LIN {X 0,Y 204.515,Z 531.386,A -85,B 0,C 180,E1 -21351.152,E2 -21351.152} C_VEL
LIN {X 0,Y 207.407,Z 525.139,A -85,B 0,C 180,E1 -21353.993,E2 -21353.993} C_VEL
LIN {X 0,Y 210.889,Z 517.359,A -85,B 0,C 180,E1 -21356.738,E2 -21356.738} C_VEL
LIN {X 0,Y 215.007,Z 507.662,A -85,B 0,C 180,E1 -21359.362,E2 -21359.362} C_VEL
LIN {X 0,Y 218.777,Z 497.655,A -85,B 0,C 180,E1 -21361.468,E2 -21361.468} C_VEL
LIN {X 0,Y 222.468,Z 486.343,A -85,B 0,C 180,E1 -21363.292,E2 -21363.292} C_VEL
LIN {X 0,Y 225.481,Z 475.279,A -85,B 0,C 180,E1 -21364.67,E2 -21364.67} C_VEL
LIN {X 0,Y 228.235,Z 462.981,A -85,B 0,C 180,E1 -21365.808,E2 -21365.808} C_VEL
LIN {X 0,Y 230.361,Z 449.627,A -85,B 0,C 180,E1 -21366.668,E2 -21366.668} C_VEL
LIN {X 0,Y 231.622,Z 436.111,A -85,B 0,C 180,E1 -21367.225,E2 -21367.225} C_VEL
LIN {X 0,Y 233.764,Z 396.806,A -85,B 0,C 180,E1 -21368.36,E2 -21368.36} C_VEL
LIN {X 0,Y 232.42,Z 387.33,A -85,B 0,C 180,E1 -21369.056,E2 -21369.056} C_VEL
LIN {X 0,Y 225.93,Z 372.695,A -85,B 0,C 180,E1 -21371.264,E2 -21371.264} C_VEL
LIN {X 0,Y 220.547,Z 361.907,A -85,B 0,C 180,E1 -21373.205,E2 -21373.205} C_VEL
LIN {X 0,Y 214.552,Z 351.494,A -85,B 0,C 180,E1 -21375.499,E2 -21375.499} C_VEL
LIN {X 0,Y 211.348,Z 346.333,A -85,B 0,C 180,E1 -21376.806,E2 -21376.806} C_VEL
LIN {X 0,Y 208.889,Z 342.383,A -85,B 0,C 180,E1 -21377.864,E2 -21377.864} C_VEL
LIN {X 0,Y 205.735,Z 337.482,A -85,B 0,C 180,E1 -21379.288,E2 -21379.288} C_VEL
LIN {X 0,Y 202.102,Z 332.43,A -85,B 0,C 180,E1 -21381.013,E2 -21381.013} C_VEL
LIN {X 0,Y 201.403,Z 331.069,A -85,B 0,C 180,E1 -21381.409,E2 -21381.409} C_VEL
LIN {X 0,Y 199.624,Z 325.609,A -85,B 0,C 180,E1 -21385.915,E2 -21385.915} C_VEL
LIN {X 0,Y 199.703,Z 325.607,A -85,B 0,C 180,E1 -21388.137,E2 -21388.137} C_VEL
LIN {X 0,Y 199.689,Z 325.602,A -85,B 0,C 180,E1 -21392.772,E2 -21392.772} C_VEL
LIN {X 0,Y 199.74,Z 325.594,A -85,B 0,C 180,E1 -21397.229,E2 -21397.229} C_VEL
LIN {X 0,Y 199.799,Z 325.585,A -85,B 0,C 180,E1 -21401.758,E2 -21401.758} C_VEL
LIN {X 0,Y 199.837,Z 325.578,A -85,B 0,C 180,E1 -21405.748,E2 -21405.748} C_VEL
LIN {X 0,Y 200.025,Z 325.552,A -85,B 0,C 180,E1 -21409.882,E2 -21409.882} C_VEL
LIN {X 0,Y 200.028,Z 325.551,A -85,B 0,C 180,E1 -21413.949,E2 -21413.949} C_VEL
LIN {X 0,Y 200.322,Z 325.516,A -85,B 0,C 180,E1 -21417.989,E2 -21417.989} C_VEL
LIN {X 0,Y 200.477,Z 325.497,A -85,B 0,C 180,E1 -21420,E2 -21420} C_VEL
LIN {X 0,Y 200.03,Z 325.551,A -85,B 0,C 180,E1 -21424.029,E2 -21424.029} C_VEL
LIN {X 0,Y 200.113,Z 325.542,A -85,B 0,C 180,E1 -21428.075,E2 -21428.075} C_VEL
LIN {X 0,Y 199.888,Z 325.573,A -85,B 0,C 180,E1 -21432.178,E2 -21432.178} C_VEL
LIN {X 0,Y 199.806,Z 325.585,A -85,B 0,C 180,E1 -21436.343,E2 -21436.343} C_VEL
LIN {X 0,Y 199.683,Z 325.601,A -85,B 0,C 180,E1 -21440.607,E2 -21440.607} C_VEL
LIN {X 0,Y 199.666,Z 325.602,A -85,B 0,C 180,E1 -21444.985,E2 -21444.985} C_VEL
LIN {X 0,Y 199.734,Z 325.752,A -85,B 0,C 180,E1 -21448.121,E2 -21448.121} C_VEL
LIN {X 0,Y 200.576,Z 328.258,A -85,B 0,C 180,E1 -21448.644,E2 -21448.644} C_VEL
LIN {X 0,Y 202.593,Z 330.528,A -85,B 0,C 180,E1 -21449.626,E2 -21449.626} C_VEL
LIN {X 0,Y 203.757,Z 331.505,A -85,B 0,C 180,E1 -21450.151,E2 -21450.151} C_VEL
LIN {X 0,Y 205.771,Z 334.706,A -85,B 0,C 180,E1 -21451.119,E2 -21451.119} C_VEL
LIN {X 0,Y 207.562,Z 336.578,A -85,B 0,C 180,E1 -21451.892,E2 -21451.892} C_VEL
LIN {X 0,Y 210.056,Z 340.063,A -85,B 0,C 180,E1 -21452.971,E2 -21452.971} C_VEL
LIN {X 0,Y 214.72,Z 346.555,A -85,B 0,C 180,E1 -21454.856,E2 -21454.856} C_VEL
LIN {X 0,Y 219.685,Z 353.753,A -85,B 0,C 180,E1 -21456.715,E2 -21456.715} C_VEL
LIN {X 0,Y 225.74,Z 363.533,A -85,B 0,C 180,E1 -21458.831,E2 -21458.831} C_VEL
LIN {X 0,Y 232.139,Z 376.228,A -85,B 0,C 180,E1 -21460.968,E2 -21460.968} C_VEL
LIN {X 0,Y 234.533,Z 381.512,A -85,B 0,C 180,E1 -21461.74,E2 -21461.74} C_VEL
LIN {X 0,Y 231.79,Z 428.656,A -85,B 0,C 180,E1 -21463.116,E2 -21463.116} C_VEL
LIN {X 0,Y 230.216,Z 442.417,A -85,B 0,C 180,E1 -21463.844,E2 -21463.844} C_VEL
LIN {X 0,Y 228.641,Z 451.728,A -85,B 0,C 180,E1 -21464.541,E2 -21464.541} C_VEL
LIN {X 0,Y 226.135,Z 464.233,A -85,B 0,C 180,E1 -21465.841,E2 -21465.841} C_VEL
LIN {X 0,Y 223.103,Z 475.556,A -85,B 0,C 180,E1 -21467.368,E2 -21467.368} C_VEL
LIN {X 0,Y 219.686,Z 486.517,A -85,B 0,C 180,E1 -21469.321,E2 -21469.321} C_VEL
LIN {X 0,Y 216.012,Z 496.198,A -85,B 0,C 180,E1 -21471.482,E2 -21471.482} C_VEL
LIN {X 0,Y 212.318,Z 504.996,A -85,B 0,C 180,E1 -21474.016,E2 -21474.016} C_VEL
LIN {X 0,Y 208.772,Z 512.595,A -85,B 0,C 180,E1 -21476.836,E2 -21476.836} C_VEL
LIN {X 0,Y 206.187,Z 517.74,A -85,B 0,C 180,E1 -21479.25,E2 -21479.25} C_VEL
LIN {X 0,Y 203.548,Z 522.69,A -85,B 0,C 180,E1 -21482.216,E2 -21482.216} C_VEL
LIN {X 0,Y 201.43,Z 526.468,A -85,B 0,C 180,E1 -21485.248,E2 -21485.248} C_VEL
LIN {X 0,Y 200.26,Z 528.4,A -85,B 0,C 180,E1 -21487.291,E2 -21487.291} C_VEL
LIN {X 0,Y 199.284,Z 529.888,A -85,B 0,C 180,E1 -21489.349,E2 -21489.349} C_VEL
LIN {X 0,Y 198.034,Z 531.536,A -85,B 0,C 180,E1 -21493.505,E2 -21493.505} C_VEL
LIN {X 0,Y 197.561,Z 531.773,A -85,B 0,C 180,E1 -21495.58,E2 -21495.58} C_VEL
LIN {X 0,Y 197.267,Z 531.587,A -85,B 0,C 180,E1 -21497.656,E2 -21497.656} C_VEL
LIN {X 0,Y 197.167,Z 530.979,A -85,B 0,C 180,E1 -21499.733,E2 -21499.733} C_VEL
LIN {X 0,Y 197.226,Z 529.981,A -85,B 0,C 180,E1 -21501.804,E2 -21501.804} C_VEL
LIN {X 0,Y 197.582,Z 527.742,A -85,B 0,C 180,E1 -21504.848,E2 -21504.848} C_VEL
LIN {X 0,Y 197.986,Z 524.459,A -85,B 0,C 180,E1 -21507.965,E2 -21507.965} C_VEL
LIN {X 0,Y 198.777,Z 520.154,A -85,B 0,C 180,E1 -21511.012,E2 -21511.012} C_VEL
LIN {X 0,Y 199.894,Z 514.673,A -85,B 0,C 180,E1 -21514.031,E2 -21514.031} C_VEL
LIN {X 0,Y 201.479,Z 507.83,A -85,B 0,C 180,E1 -21517.011,E2 -21517.011} C_VEL
LIN {X 0,Y 203.48,Z 499.275,A -85,B 0,C 180,E1 -21519.943,E2 -21519.943} C_VEL
LIN {X 0,Y 205.467,Z 490.5,A -85,B 0,C 180,E1 -21522.343,E2 -21522.343} C_VEL
LIN {X 0,Y 207.813,Z 479.69,A -85,B 0,C 180,E1 -21524.692,E2 -21524.692} C_VEL
LIN {X 0,Y 210.013,Z 468.775,A -85,B 0,C 180,E1 -21526.525,E2 -21526.525} C_VEL
LIN {X 0,Y 211.732,Z 458.541,A -85,B 0,C 180,E1 -21527.879,E2 -21527.879} C_VEL
LIN {X 0,Y 213.036,Z 446.448,A -85,B 0,C 180,E1 -21529.136,E2 -21529.136} C_VEL
LIN {X 0,Y 214.045,Z 434.997,A -85,B 0,C 180,E1 -21529.978,E2 -21529.978} C_VEL
LIN {X 0,Y 215.03,Z 421.503,A -85,B 0,C 180,E1 -21530.569,E2 -21530.569} C_VEL
LIN {X 0,Y 217.234,Z 363.666,A -85,B 0,C 180,E1 -21532.399,E2 -21532.399} C_VEL
LIN {X 0,Y 212.328,Z 350.513,A -85,B 0,C 180,E1 -21533.621,E2 -21533.621} C_VEL
LIN {X 0,Y 204.773,Z 335.543,A -85,B 0,C 180,E1 -21535.433,E2 -21535.433} C_VEL
LIN {X 0,Y 200.996,Z 328.962,A -85,B 0,C 180,E1 -21536.366,E2 -21536.366} C_VEL
LIN {X 0,Y 199.845,Z 326.586,A -85,B 0,C 180,E1 -21536.674,E2 -21536.674} C_VEL
LIN {X 0,Y 199.667,Z 325.605,A -85,B 0,C 180,E1 -21536.794,E2 -21536.794} C_VEL
LIN {X 0,Y 199.663,Z 325.612,A -85,B 0,C 180,E1 -21542.351,E2 -21542.351} C_VEL
LIN {X 0,Y 199.616,Z 325.618,A -85,B 0,C 180,E1 -21546.763,E2 -21546.763} C_VEL
LIN {X 0,Y 199.591,Z 325.617,A -85,B 0,C 180,E1 -21549.33,E2 -21549.33} C_VEL
LIN {X 0,Y 199.562,Z 325.625,A -85,B 0,C 180,E1 -21552.306,E2 -21552.306} C_VEL
LIN {X 0,Y 199.572,Z 325.614,A -85,B 0,C 180,E1 -21555.227,E2 -21555.227} C_VEL
LIN {X 0,Y 199.573,Z 325.622,A -85,B 0,C 180,E1 -21558.003,E2 -21558.003} C_VEL
LIN {X 0,Y 199.605,Z 325.605,A -85,B 0,C 180,E1 -21560.767,E2 -21560.767} C_VEL
LIN {X 0,Y 199.607,Z 325.619,A -85,B 0,C 180,E1 -21565.713,E2 -21565.713} C_VEL
LIN {X 0,Y 199.688,Z 325.599,A -85,B 0,C 180,E1 -21568.135,E2 -21568.135} C_VEL
LIN {X 0,Y 199.68,Z 325.606,A -85,B 0,C 180,E1 -21572.771,E2 -21572.771} C_VEL
LIN {X 0,Y 199.708,Z 325.6,A -85,B 0,C 180,E1 -21577.226,E2 -21577.226} C_VEL
LIN {X 0,Y 199.79,Z 325.586,A -85,B 0,C 180,E1 -21581.758,E2 -21581.758} C_VEL
LIN {X 0,Y 199.83,Z 325.594,A -85,B 0,C 180,E1 -21585.748,E2 -21585.748} C_VEL
LIN {X 0,Y 200.017,Z 325.547,A -85,B 0,C 180,E1 -21589.882,E2 -21589.882} C_VEL
LIN {X 0,Y 200.009,Z 325.568,A -85,B 0,C 180,E1 -21593.949,E2 -21593.949} C_VEL
LIN {X 0,Y 200.313,Z 325.525,A -85,B 0,C 180,E1 -21597.99,E2 -21597.99} C_VEL
LIN {X 0,Y 200.47,Z 325.492,A -85,B 0,C 180,E1 -21600,E2 -21600} C_VEL
LIN {X 0,Y 200.023,Z 325.564,A -85,B 0,C 180,E1 -21604.03,E2 -21604.03} C_VEL
LIN {X 0,Y 200.105,Z 325.554,A -85,B 0,C 180,E1 -21608.076,E2 -21608.076} C_VEL
LIN {X 0,Y 200.031,Z 325.547,A -85,B 0,C 180,E1 -21610.348,E2 -21610.348} C_VEL
LIN {X 0,Y 199.799,Z 325.597,A -85,B 0,C 180,E1 -21616.344,E2 -21616.344} C_VEL
LIN {X 0,Y 199.695,Z 325.611,A -85,B 0,C 180,E1 -21620.606,E2 -21620.606} C_VEL
LIN {X 0,Y 199.668,Z 325.614,A -85,B 0,C 180,E1 -21624.985,E2 -21624.985} C_VEL
LIN {X 0,Y 199.671,Z 325.612,A -85,B 0,C 180,E1 -21629.523,E2 -21629.523} C_VEL
LIN {X 0,Y 199.66,Z 325.616,A -85,B 0,C 180,E1 -21632.353,E2 -21632.353} C_VEL
LIN {X 0,Y 199.637,Z 325.618,A -85,B 0,C 180,E1 -21636.761,E2 -21636.761} C_VEL
LIN {X 0,Y 199.636,Z 325.62,A -85,B 0,C 180,E1 -21639.322,E2 -21639.322} C_VEL
LIN {X 0,Y 199.574,Z 325.627,A -85,B 0,C 180,E1 -21644.773,E2 -21644.773} C_VEL
LIN {X 0,Y 199.67,Z 325.772,A -85,B 0,C 180,E1 -21649.666,E2 -21649.666} C_VEL
LIN {X 0,Y 201.559,Z 333.298,A -85,B 0,C 180,E1 -21653.412,E2 -21653.412} C_VEL
LIN {X 0,Y 209.685,Z 352.389,A -85,B 0,C 180,E1 -21655.541,E2 -21655.541} C_VEL
LIN {X 0,Y 210.618,Z 354.668,A -85,B 0,C 180,E1 -21655.775,E2 -21655.775} C_VEL
LIN {X 0,Y 211.311,Z 357.711,A -85,B 0,C 180,E1 -21656,E2 -21656} C_VEL
LIN {X 0,Y 210.901,Z 362.309,A -85,B 0,C 180,E1 -21656.114,E2 -21656.114} C_VEL
LIN {X 0,Y 208.654,Z 371.718,A -85,B 0,C 180,E1 -21656.131,E2 -21656.131} C_VEL
LIN {X 0,Y 208.592,Z 375.791,A -85,B 0,C 180,E1 -21656.28,E2 -21656.28} C_VEL
LIN {X 0,Y 210.096,Z 391.661,A -85,B 0,C 180,E1 -21657.118,E2 -21657.118} C_VEL
LIN {X 0,Y 207.932,Z 442.645,A -85,B 0,C 180,E1 -21658.821,E2 -21658.821} C_VEL
LIN {X 0,Y 206.586,Z 456.624,A -85,B 0,C 180,E1 -21659.672,E2 -21659.672} C_VEL
LIN {X 0,Y 204.839,Z 469.498,A -85,B 0,C 180,E1 -21660.873,E2 -21660.873} C_VEL
LIN {X 0,Y 202.798,Z 481.278,A -85,B 0,C 180,E1 -21662.388,E2 -21662.388} C_VEL
LIN {X 0,Y 200.405,Z 492.63,A -85,B 0,C 180,E1 -21664.281,E2 -21664.281} C_VEL
LIN {X 0,Y 198.123,Z 502.854,A -85,B 0,C 180,E1 -21666.481,E2 -21666.481} C_VEL
LIN {X 0,Y 195.942,Z 512.061,A -85,B 0,C 180,E1 -21668.983,E2 -21668.983} C_VEL
LIN {X 0,Y 194.595,Z 518.294,A -85,B 0,C 180,E1 -21671.033,E2 -21671.033} C_VEL
LIN {X 0,Y 192.786,Z 525.982,A -85,B 0,C 180,E1 -21674.134,E2 -21674.134} C_VEL
LIN {X 0,Y 191.457,Z 532.154,A -85,B 0,C 180,E1 -21677.278,E2 -21677.278} C_VEL
LIN {X 0,Y 190.689,Z 537.042,A -85,B 0,C 180,E1 -21680.455,E2 -21680.455} C_VEL
LIN {X 0,Y 190.346,Z 540.785,A -85,B 0,C 180,E1 -21683.642,E2 -21683.642} C_VEL
LIN {X 0,Y 190.236,Z 542.851,A -85,B 0,C 180,E1 -21685.934,E2 -21685.934} C_VEL
LIN {X 0,Y 190.27,Z 544.186,A -85,B 0,C 180,E1 -21687.884,E2 -21687.884} C_VEL
LIN {X 0,Y 190.407,Z 545.217,A -85,B 0,C 180,E1 -21690.001,E2 -21690.001} C_VEL
LIN {X 0,Y 190.16,Z 546.04,A -85,B 0,C 180,E1 -21693.729,E2 -21693.729} C_VEL
LIN {X 0,Y 190.281,Z 545.91,A -85,B 0,C 180,E1 -21696.363,E2 -21696.363} C_VEL
LIN {X 0,Y 191.021,Z 544.357,A -85,B 0,C 180,E1 -21700.601,E2 -21700.601} C_VEL
LIN {X 0,Y 192.552,Z 541.238,A -85,B 0,C 180,E1 -21704.804,E2 -21704.804} C_VEL
LIN {X 0,Y 194.5,Z 537.748,A -85,B 0,C 180,E1 -21707.888,E2 -21707.888} C_VEL
LIN {X 0,Y 196.934,Z 533.191,A -85,B 0,C 180,E1 -21710.909,E2 -21710.909} C_VEL
LIN {X 0,Y 199.958,Z 527.201,A -85,B 0,C 180,E1 -21713.959,E2 -21713.959} C_VEL
LIN {X 0,Y 203.267,Z 520.26,A -85,B 0,C 180,E1 -21716.711,E2 -21716.711} C_VEL
LIN {X 0,Y 207.388,Z 511.367,A -85,B 0,C 180,E1 -21719.432,E2 -21719.432} C_VEL
LIN {X 0,Y 211.146,Z 502.261,A -85,B 0,C 180,E1 -21721.618,E2 -21721.618} C_VEL
LIN {X 0,Y 214.85,Z 492.184,A -85,B 0,C 180,E1 -21723.505,E2 -21723.505} C_VEL
LIN {X 0,Y 218.377,Z 481.017,A -85,B 0,C 180,E1 -21725.119,E2 -21725.119} C_VEL
LIN {X 0,Y 221.118,Z 470.477,A -85,B 0,C 180,E1 -21726.298,E2 -21726.298} C_VEL
LIN {X 0,Y 223.638,Z 458.434,A -85,B 0,C 180,E1 -21727.299,E2 -21727.299} C_VEL
LIN {X 0,Y 225.45,Z 445.983,A -85,B 0,C 180,E1 -21728.029,E2 -21728.029} C_VEL
LIN {X 0,Y 226.704,Z 430.015,A -85,B 0,C 180,E1 -21728.584,E2 -21728.584} C_VEL
LIN {X 0,Y 228.506,Z 397.917,A -85,B 0,C 180,E1 -21729.526,E2 -21729.526} C_VEL
LIN {X 0,Y 227.385,Z 390.224,A -85,B 0,C 180,E1 -21730.129,E2 -21730.129} C_VEL
LIN {X 0,Y 221.007,Z 375.641,A -85,B 0,C 180,E1 -21732.433,E2 -21732.433} C_VEL
LIN {X 0,Y 215.831,Z 365.308,A -85,B 0,C 180,E1 -21734.411,E2 -21734.411} C_VEL
LIN {X 0,Y 210.412,Z 355.756,A -85,B 0,C 180,E1 -21736.618,E2 -21736.618} C_VEL
LIN {X 0,Y 205.54,Z 347.769,A -85,B 0,C 180,E1 -21738.769,E2 -21738.769} C_VEL
LIN {X 0,Y 201.701,Z 341.932,A -85,B 0,C 180,E1 -21740.594,E2 -21740.594} C_VEL
LIN {X 0,Y 198.13,Z 336.598,A -85,B 0,C 180,E1 -21742.434,E2 -21742.434} C_VEL
LIN {X 0,Y 194.41,Z 331.564,A -85,B 0,C 180,E1 -21744.497,E2 -21744.497} C_VEL
LIN {X 0,Y 193.891,Z 330.514,A -85,B 0,C 180,E1 -21744.871,E2 -21744.871} C_VEL
LIN {X 0,Y 192.635,Z 326.482,A -85,B 0,C 180,E1 -21748.675,E2 -21748.675} C_VEL
LIN {X 0,Y 192.667,Z 326.485,A -85,B 0,C 180,E1 -21751.692,E2 -21751.692} C_VEL
LIN {X 0,Y 192.708,Z 326.473,A -85,B 0,C 180,E1 -21756.349,E2 -21756.349} C_VEL
LIN {X 0,Y 192.734,Z 326.465,A -85,B 0,C 180,E1 -21761.458,E2 -21761.458} C_VEL
LIN {X 0,Y 192.766,Z 326.459,A -85,B 0,C 180,E1 -21765.214,E2 -21765.214} C_VEL
LIN {X 0,Y 192.947,Z 326.434,A -85,B 0,C 180,E1 -21769.566,E2 -21769.566} C_VEL
LIN {X 0,Y 193.043,Z 326.43,A -85,B 0,C 180,E1 -21771.626,E2 -21771.626} C_VEL
LIN {X 0,Y 193.264,Z 326.395,A -85,B 0,C 180,E1 -21777.916,E2 -21777.916} C_VEL
LIN {X 0,Y 193.442,Z 326.373,A -85,B 0,C 180,E1 -21780,E2 -21780} C_VEL
LIN {X 0,Y 192.977,Z 326.43,A -85,B 0,C 180,E1 -21784.177,E2 -21784.177} C_VEL
LIN {X 0,Y 193.064,Z 326.42,A -85,B 0,C 180,E1 -21788.372,E2 -21788.372} C_VEL
LIN {X 0,Y 192.811,Z 326.454,A -85,B 0,C 180,E1 -21792.632,E2 -21792.632} C_VEL
LIN {X 0,Y 192.759,Z 326.463,A -85,B 0,C 180,E1 -21796.958,E2 -21796.958} C_VEL
LIN {X 0,Y 192.617,Z 326.482,A -85,B 0,C 180,E1 -21801.399,E2 -21801.399} C_VEL
LIN {X 0,Y 192.624,Z 326.479,A -85,B 0,C 180,E1 -21804.773,E2 -21804.773} C_VEL
LIN {X 0,Y 193.469,Z 329.055,A -85,B 0,C 180,E1 -21805.412,E2 -21805.412} C_VEL
LIN {X 0,Y 195.274,Z 331.189,A -85,B 0,C 180,E1 -21806.448,E2 -21806.448} C_VEL
LIN {X 0,Y 196.904,Z 332.299,A -85,B 0,C 180,E1 -21807.285,E2 -21807.285} C_VEL
LIN {X 0,Y 198.681,Z 335.411,A -85,B 0,C 180,E1 -21808.284,E2 -21808.284} C_VEL
LIN {X 0,Y 201.002,Z 337.731,A -85,B 0,C 180,E1 -21809.416,E2 -21809.416} C_VEL
LIN {X 0,Y 203.486,Z 341.24,A -85,B 0,C 180,E1 -21810.626,E2 -21810.626} C_VEL
LIN {X 0,Y 204.83,Z 342.917,A -85,B 0,C 180,E1 -21811.241,E2 -21811.241} C_VEL
LIN {X 0,Y 210.653,Z 350.923,A -85,B 0,C 180,E1 -21813.759,E2 -21813.759} C_VEL
LIN {X 0,Y 217.978,Z 362.001,A -85,B 0,C 180,E1 -21816.618,E2 -21816.618} C_VEL
LIN {X 0,Y 223.149,Z 371.017,A -85,B 0,C 180,E1 -21818.486,E2 -21818.486} C_VEL
LIN {X 0,Y 229.249,Z 383.852,A -85,B 0,C 180,E1 -21820.603,E2 -21820.603} C_VEL
LIN {X 0,Y 226.489,Z 429.139,A -85,B 0,C 180,E1 -21821.947,E2 -21821.947} C_VEL
LIN {X 0,Y 224.904,Z 442.518,A -85,B 0,C 180,E1 -21822.665,E2 -21822.665} C_VEL
LIN {X 0,Y 223.142,Z 452.442,A -85,B 0,C 180,E1 -21823.417,E2 -21823.417} C_VEL
LIN {X 0,Y 220.671,Z 464.314,A -85,B 0,C 180,E1 -21824.676,E2 -21824.676} C_VEL
LIN {X 0,Y 217.802,Z 474.69,A -85,B 0,C 180,E1 -21826.071,E2 -21826.071} C_VEL
LIN {X 0,Y 214.59,Z 484.804,A -85,B 0,C 180,E1 -21827.825,E2 -21827.825} C_VEL
LIN {X 0,Y 211.006,Z 494.248,A -85,B 0,C 180,E1 -21829.883,E2 -21829.883} C_VEL
LIN {X 0,Y 207.117,Z 503.2,A -85,B 0,C 180,E1 -21832.353,E2 -21832.353} C_VEL
LIN {X 0,Y 203.27,Z 511.259,A -85,B 0,C 180,E1 -21835.215,E2 -21835.215} C_VEL
LIN {X 0,Y 199.953,Z 517.635,A -85,B 0,C 180,E1 -21838.181,E2 -21838.181} C_VEL
LIN {X 0,Y 197.122,Z 522.665,A -85,B 0,C 180,E1 -21841.228,E2 -21841.228} C_VEL
LIN {X 0,Y 194.763,Z 526.61,A -85,B 0,C 180,E1 -21844.438,E2 -21844.438} C_VEL
LIN {X 0,Y 193.558,Z 528.486,A -85,B 0,C 180,E1 -21846.458,E2 -21846.458} C_VEL
LIN {X 0,Y 192.473,Z 530.026,A -85,B 0,C 180,E1 -21848.583,E2 -21848.583} C_VEL
LIN {X 0,Y 191.642,Z 531.1,A -85,B 0,C 180,E1 -21850.727,E2 -21850.727} C_VEL
LIN {X 0,Y 190.998,Z 531.799,A -85,B 0,C 180,E1 -21853.077,E2 -21853.077} C_VEL
LIN {X 0,Y 190.23,Z 531.899,A -85,B 0,C 180,E1 -21857.192,E2 -21857.192} C_VEL
LIN {X 0,Y 190.096,Z 531.328,A -85,B 0,C 180,E1 -21859.346,E2 -21859.346} C_VEL
LIN {X 0,Y 190.117,Z 530.363,A -85,B 0,C 180,E1 -21861.496,E2 -21861.496} C_VEL
LIN {X 0,Y 190.492,Z 527.934,A -85,B 0,C 180,E1 -21864.958,E2 -21864.958} C_VEL
LIN {X 0,Y 190.895,Z 524.974,A -85,B 0,C 180,E1 -21867.889,E2 -21867.889} C_VEL
LIN {X 0,Y 191.68,Z 520.745,A -85,B 0,C 180,E1 -21871.049,E2 -21871.049} C_VEL
LIN {X 0,Y 193.039,Z 514.339,A -85,B 0,C 180,E1 -21874.698,E2 -21874.698} C_VEL
LIN {X 0,Y 194.763,Z 507.33,A -85,B 0,C 180,E1 -21877.776,E2 -21877.776} C_VEL
LIN {X 0,Y 196.909,Z 498.569,A -85,B 0,C 180,E1 -21880.799,E2 -21880.799} C_VEL
LIN {X 0,Y 199.26,Z 488.625,A -85,B 0,C 180,E1 -21883.512,E2 -21883.512} C_VEL
LIN {X 0,Y 201.506,Z 478.459,A -85,B 0,C 180,E1 -21885.681,E2 -21885.681} C_VEL
LIN {X 0,Y 203.87,Z 467.146,A -85,B 0,C 180,E1 -21887.555,E2 -21887.555} C_VEL
LIN {X 0,Y 205.672,Z 455.483,A -85,B 0,C 180,E1 -21889.071,E2 -21889.071} C_VEL
LIN {X 0,Y 206.997,Z 442.814,A -85,B 0,C 180,E1 -21890.299,E2 -21890.299} C_VEL
LIN {X 0,Y 208.033,Z 431.473,A -85,B 0,C 180,E1 -21891.034,E2 -21891.034} C_VEL
LIN {X 0,Y 209.135,Z 413.294,A -85,B 0,C 180,E1 -21891.693,E2 -21891.693} C_VEL
LIN {X 0,Y 210.984,Z 365.325,A -85,B 0,C 180,E1 -21893.258,E2 -21893.258} C_VEL
LIN {X 0,Y 206.449,Z 353.278,A -85,B 0,C 180,E1 -21894.443,E2 -21894.443} C_VEL
LIN {X 0,Y 198.173,Z 336.981,A -85,B 0,C 180,E1 -21896.544,E2 -21896.544} C_VEL
LIN {X 0,Y 193.851,Z 329.708,A -85,B 0,C 180,E1 -21897.679,E2 -21897.679} C_VEL
LIN {X 0,Y 192.669,Z 326.877,A -85,B 0,C 180,E1 -21898.038,E2 -21898.038} C_VEL
LIN {X 0,Y 192.632,Z 326.486,A -85,B 0,C 180,E1 -21898.117,E2 -21898.117} C_VEL
LIN {X 0,Y 192.592,Z 326.494,A -85,B 0,C 180,E1 -21903.185,E2 -21903.185} C_VEL
LIN {X 0,Y 192.539,Z 326.492,A -85,B 0,C 180,E1 -21908.353,E2 -21908.353} C_VEL
LIN {X 0,Y 192.48,Z 326.498,A -85,B 0,C 180,E1 -21913.092,E2 -21913.092} C_VEL
LIN {X 0,Y 192.485,Z 326.505,A -85,B 0,C 180,E1 -21916.904,E2 -21916.904} C_VEL
LIN {X 0,Y 192.546,Z 326.482,A -85,B 0,C 180,E1 -21921.647,E2 -21921.647} C_VEL
LIN {X 0,Y 192.592,Z 326.492,A -85,B 0,C 180,E1 -21926.813,E2 -21926.813} C_VEL
LIN {X 0,Y 192.655,Z 326.473,A -85,B 0,C 180,E1 -21931.691,E2 -21931.691} C_VEL
LIN {X 0,Y 192.68,Z 326.48,A -85,B 0,C 180,E1 -21936.345,E2 -21936.345} C_VEL
LIN {X 0,Y 192.725,Z 326.463,A -85,B 0,C 180,E1 -21941.459,E2 -21941.459} C_VEL
LIN {X 0,Y 192.758,Z 326.473,A -85,B 0,C 180,E1 -21945.214,E2 -21945.214} C_VEL
LIN {X 0,Y 192.939,Z 326.428,A -85,B 0,C 180,E1 -21949.567,E2 -21949.567} C_VEL
LIN {X 0,Y 192.971,Z 326.443,A -85,B 0,C 180,E1 -21953.728,E2 -21953.728} C_VEL
LIN {X 0,Y 193.255,Z 326.404,A -85,B 0,C 180,E1 -21957.916,E2 -21957.916} C_VEL
LIN {X 0,Y 193.434,Z 326.367,A -85,B 0,C 180,E1 -21960,E2 -21960} C_VEL
LIN {X 0,Y 192.97,Z 326.443,A -85,B 0,C 180,E1 -21964.177,E2 -21964.177} C_VEL
LIN {X 0,Y 193.056,Z 326.428,A -85,B 0,C 180,E1 -21968.373,E2 -21968.373} C_VEL
LIN {X 0,Y 192.804,Z 326.453,A -85,B 0,C 180,E1 -21972.634,E2 -21972.634} C_VEL
LIN {X 0,Y 192.752,Z 326.473,A -85,B 0,C 180,E1 -21976.959,E2 -21976.959} C_VEL
LIN {X 0,Y 192.631,Z 326.487,A -85,B 0,C 180,E1 -21981.398,E2 -21981.398} C_VEL
LIN {X 0,Y 192.66,Z 326.487,A -85,B 0,C 180,E1 -21984.226,E2 -21984.226} C_VEL
LIN {X 0,Y 192.646,Z 326.49,A -85,B 0,C 180,E1 -21988.893,E2 -21988.893} C_VEL
LIN {X 0,Y 192.597,Z 326.495,A -85,B 0,C 180,E1 -21993.187,E2 -21993.187} C_VEL
LIN {X 0,Y 192.571,Z 326.501,A -85,B 0,C 180,E1 -21998.348,E2 -21998.348} C_VEL
LIN {X 0,Y 192.487,Z 326.512,A -85,B 0,C 180,E1 -22003.097,E2 -22003.097} C_VEL
LIN {X 0,Y 192.564,Z 326.621,A -85,B 0,C 180,E1 -22008.694,E2 -22008.694} C_VEL
LIN {X 0,Y 194.261,Z 333.075,A -85,B 0,C 180,E1 -22012.048,E2 -22012.048} C_VEL
LIN {X 0,Y 201.459,Z 349.248,A -85,B 0,C 180,E1 -22014.053,E2 -22014.053} C_VEL
LIN {X 0,Y 207.127,Z 363.842,A -85,B 0,C 180,E1 -22015.583,E2 -22015.583} C_VEL
LIN {X 0,Y 208.592,Z 375.791,A -85,B 0,C 180,E1 -22016.28,E2 -22016.28} C_VEL
